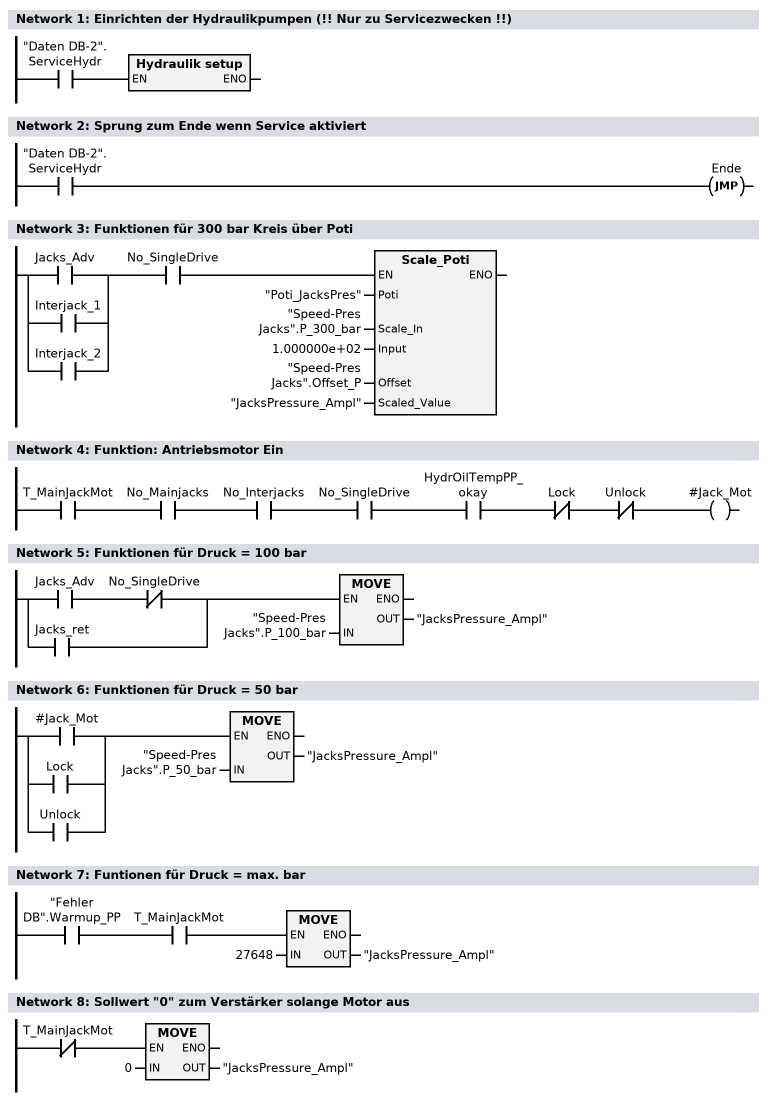
[picture p24: Jacks pressure networks 1-8]
NETWORK
TITLE = Einrichten der Hydraulikpumpen (!! Nur zu Servicezwecken !!)
      A     "Daten DB-2".ServiceHydr;
      JNB   _001;
      CALL  "Hydraulik setup";
_001: NOP   0;
NETWORK
TITLE = Sprung zum Ende wenn Service aktiviert
      A     "Daten DB-2".ServiceHydr;
      JC    Ende;
NETWORK
TITLE = Funktionen für 300 bar Kreis über Poti
      A(;
      O     "Jacks_Adv";
      O     "Interjack_1";
      O     "Interjack_2";
      );
      A     "No_SingleDrive";
      JNB   _002;
      CALL  "Scale_Poti" (
           Poti                     := "Poti_JacksPres",
           Scale_In                 := "Speed-Pres Jacks".P_300_bar,
           Input                    := 1.000000e+02,
           Offset                   := "Speed-Pres Jacks".Offset_P,
           Scaled_Value             := "JacksPressure_Ampl");
_002: NOP   0;
NETWORK
TITLE = Funktion: Antriebsmotor Ein
      A     "T_MainJackMot";
      A     "No_Mainjacks";
      A     "No_Interjacks";
      A     "No_SingleDrive";
      A     "HydrOilTempPP_okay";
      AN    "Lock";
      AN    "Unlock";
      =     #Jack_Mot;
NETWORK
TITLE = Funktionen für Druck = 100 bar
      A(;
      A     "Jacks_Adv";
      AN    "No_SingleDrive";
      O     "Jacks_ret";
      );
      JNB   _003;
      L     "Speed-Pres Jacks".P_100_bar;
      T     "JacksPressure_Ampl";
_003: NOP   0;
NETWORK
TITLE = Funktionen für Druck = 50 bar
      A(;
      O     #Jack_Mot;
      O     "Lock";
      O     "Unlock";
      );
      JNB   _004;
      L     "Speed-Pres Jacks".P_50_bar;
      T     "JacksPressure_Ampl";
_004: NOP   0;
NETWORK
TITLE = Funtionen für Druck = max. bar
      A     "Fehler DB".Warmup_PP;
      A     "T_MainJackMot";
      JNB   _005;
      L     27648;
      T     "JacksPressure_Ampl";
_005: NOP   0;
NETWORK
TITLE = Sollwert "0" zum Verstärker solange Motor aus
      AN    "T_MainJackMot";
      JNB   _006;
      L     0;
      T     "JacksPressure_Ampl";
_006: NOP   0;
NETWORK
TITLE =
Ende: NOP   0;
END_FUNCTION

FUNCTION "Cutter control" : VOID	// FC 25
TITLE = Schürfradsteuerung links/rechts
AUTHOR : Simdon
FAMILY : Cutter
NAME : Cut_Con
VERSION : 0.1
VAR_TEMP
  Mot_okay : BOOL ;	//Antriebsmotor für Hydraulik
  H_Right : BOOL ;
  H_Left : BOOL ;
END_VAR
BEGIN
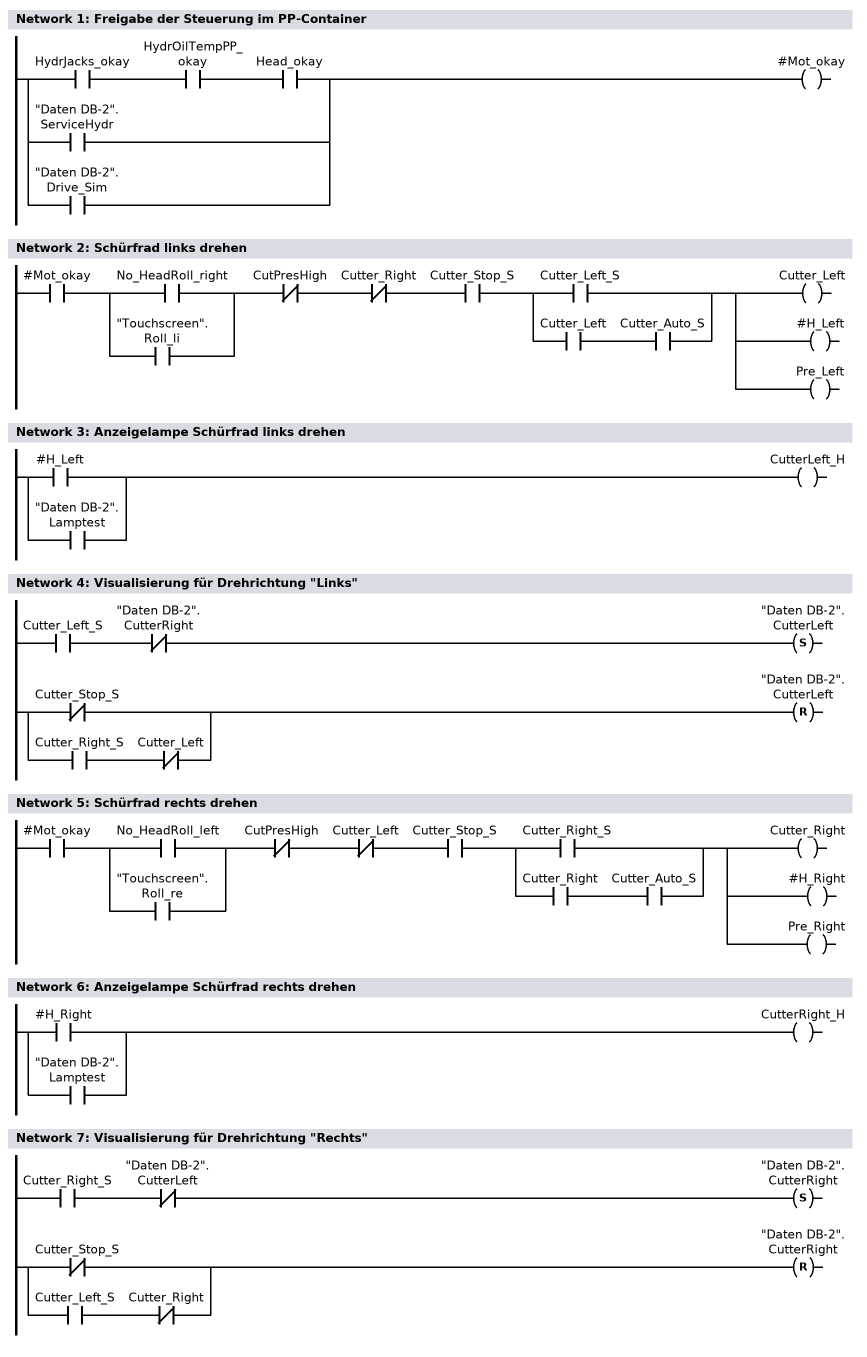
NETWORK
TITLE = Freigabe der Steuerung im PP-Container
      A     "HydrJacks_okay";
      A     "HydrOilTempPP_okay";
      A     "Head_okay";
      O     "Daten DB-2".ServiceHydr;
      O     "Daten DB-2".Drive_Sim;
      =     #Mot_okay;
NETWORK
TITLE = Schürfrad links drehen
//Schürfrad dreht in einer der gewählten Betriebsarten links herum.
      A     #Mot_okay;
      A(;
      O     "No_HeadRoll_right";
      O     "Touchscreen".Roll_li;
      );
      AN    "CutPresHigh";
      AN    "Cutter_Right";
      A     "Cutter_Stop_S";
      A(;
      O     "Cutter_Left_S";
      O;
      A     "Cutter_Left";
      A     "Cutter_Auto_S";
      );
      =     "Cutter_Left";
      =     #H_Left;
      =     "Pre_Left";
NETWORK
TITLE = Anzeigelampe Schürfrad links drehen
      O     #H_Left;
      O     "Daten DB-2".Lamptest;
      =     "CutterLeft_H";
NETWORK
TITLE = Visualisierung für Drehrichtung "Links"
      A     "Cutter_Left_S";
      AN    "Daten DB-2".CutterRight;
      S     "Daten DB-2".CutterLeft;
      A(;
      ON    "Cutter_Stop_S";
      O;
      A     "Cutter_Right_S";
      AN    "Cutter_Left";
      );
      R     "Daten DB-2".CutterLeft;
      NOP   0;
NETWORK
TITLE = Schürfrad rechts drehen
//Schürfrad dreht in einer der gewählten Betriebsarten rechts herum.
      A     #Mot_okay;
      A(;
      O     "No_HeadRoll_left";
      O     "Touchscreen".Roll_re;
      );
      AN    "CutPresHigh";
      AN    "Cutter_Left";
      A     "Cutter_Stop_S";
      A(;
      O     "Cutter_Right_S";
      O;
      A     "Cutter_Right";
      A     "Cutter_Auto_S";
      );
      =     "Cutter_Right";
      =     #H_Right;
      =     "Pre_Right";
NETWORK
TITLE = Anzeigelampe Schürfrad rechts drehen
      O     #H_Right;
      O     "Daten DB-2".Lamptest;
      =     "CutterRight_H";
NETWORK
TITLE = Visualisierung für Drehrichtung "Rechts"
      A     "Cutter_Right_S";
      AN    "Daten DB-2".CutterLeft;
      S     "Daten DB-2".CutterRight;
      A(;
      ON    "Cutter_Stop_S";
      O;
      A     "Cutter_Left_S";
      AN    "Cutter_Right";
      );
      R     "Daten DB-2".CutterRight;
      NOP   0;
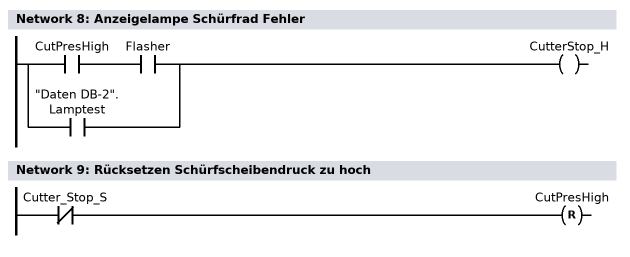
NETWORK
TITLE = Anzeigelampe Schürfrad Fehler
      A     "CutPresHigh";
      A     "Flasher";
      O     "Daten DB-2".Lamptest;
      =     "CutterStop_H";
NETWORK
TITLE = Rücksetzen Schürfscheibendruck zu hoch
      AN    "Cutter_Stop_S";
      R     "CutPresHigh";
END_FUNCTION

FUNCTION "Cutter speed" : VOID	// FC 26
TITLE = Volumenstromeinstellung für Schürfrad im PP-Container
AUTHOR : Simdon
FAMILY : Cutter
NAME : CutVol
VERSION : 0.1
VAR_TEMP
  Ltr_200 : BOOL ;
  Ltr_270 : BOOL ;
  Ltr_max : BOOL ;
END_VAR
BEGIN
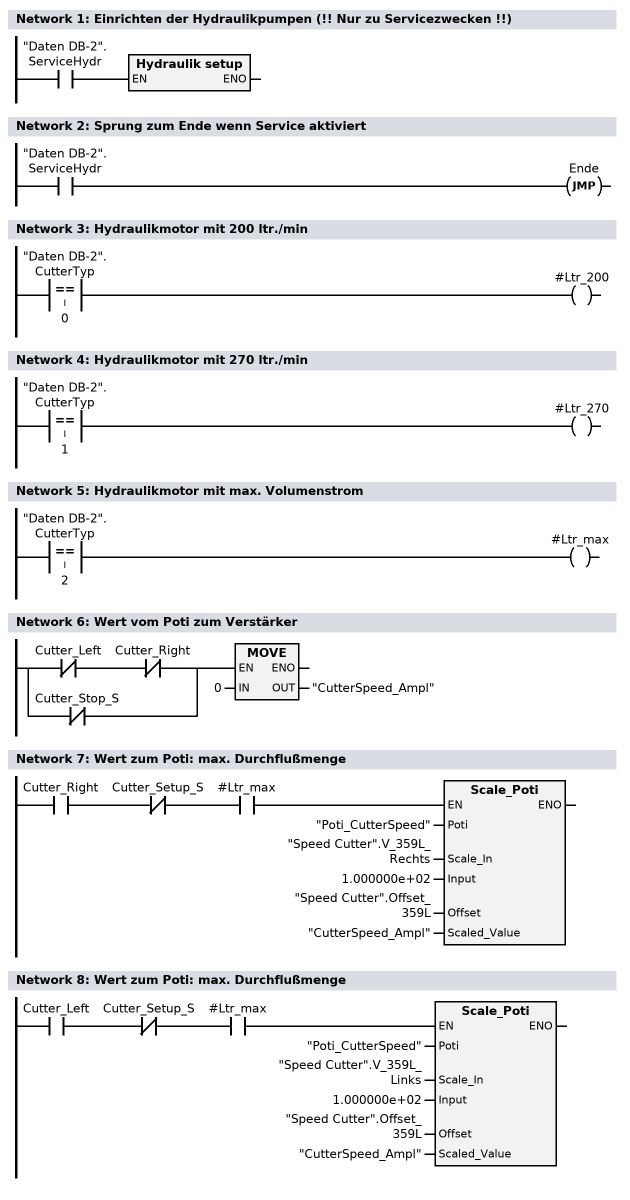
NETWORK
TITLE = Einrichten der Hydraulikpumpen (!! Nur zu Servicezwecken !!)
      A     "Daten DB-2".ServiceHydr;
      JNB   _001;
      CALL  "Hydraulik setup";
_001: NOP   0;
NETWORK
TITLE = Sprung zum Ende wenn Service aktiviert
      A     "Daten DB-2".ServiceHydr;
      JC    Ende;
NETWORK
TITLE = Hydraulikmotor mit 200 ltr./min
      L     "Daten DB-2".CutterTyp;
      L     0;
      ==I;
      =     #Ltr_200;
NETWORK
TITLE = Hydraulikmotor mit 270 ltr./min
      L     "Daten DB-2".CutterTyp;
      L     1;
      ==I;
      =     #Ltr_270;
NETWORK
TITLE = Hydraulikmotor mit max. Volumenstrom
      L     "Daten DB-2".CutterTyp;
      L     2;
      ==I;
      =     #Ltr_max;
NETWORK
TITLE = Wert vom Poti zum Verstärker
      A(;
      AN    "Cutter_Left";
      AN    "Cutter_Right";
      ON    "Cutter_Stop_S";
      );
      JNB   _002;
      L     0;
      T     "CutterSpeed_Ampl";
_002: NOP   0;
NETWORK
TITLE = Wert zum Poti: max. Durchflußmenge
      A     "Cutter_Right";
      AN    "Cutter_Setup_S";
      A     #Ltr_max;
      JNB   _003;
      CALL  "Scale_Poti" (
           Poti                     := "Poti_CutterSpeed",
           Scale_In                 := "Speed Cutter".V_359L_Rechts,
           Input                    := 1.000000e+02,
           Offset                   := "Speed Cutter".Offset_359L,
           Scaled_Value             := "CutterSpeed_Ampl");
_003: NOP   0;
NETWORK
TITLE = Wert zum Poti: max. Durchflußmenge
      A     "Cutter_Left";
      AN    "Cutter_Setup_S";
      A     #Ltr_max;
      JNB   _004;
      CALL  "Scale_Poti" (
           Poti                     := "Poti_CutterSpeed",
           Scale_In                 := "Speed Cutter".V_359L_Links,
           Input                    := 1.000000e+02,
           Offset                   := "Speed Cutter".Offset_359L,
           Scaled_Value             := "CutterSpeed_Ampl");
_004: NOP   0;
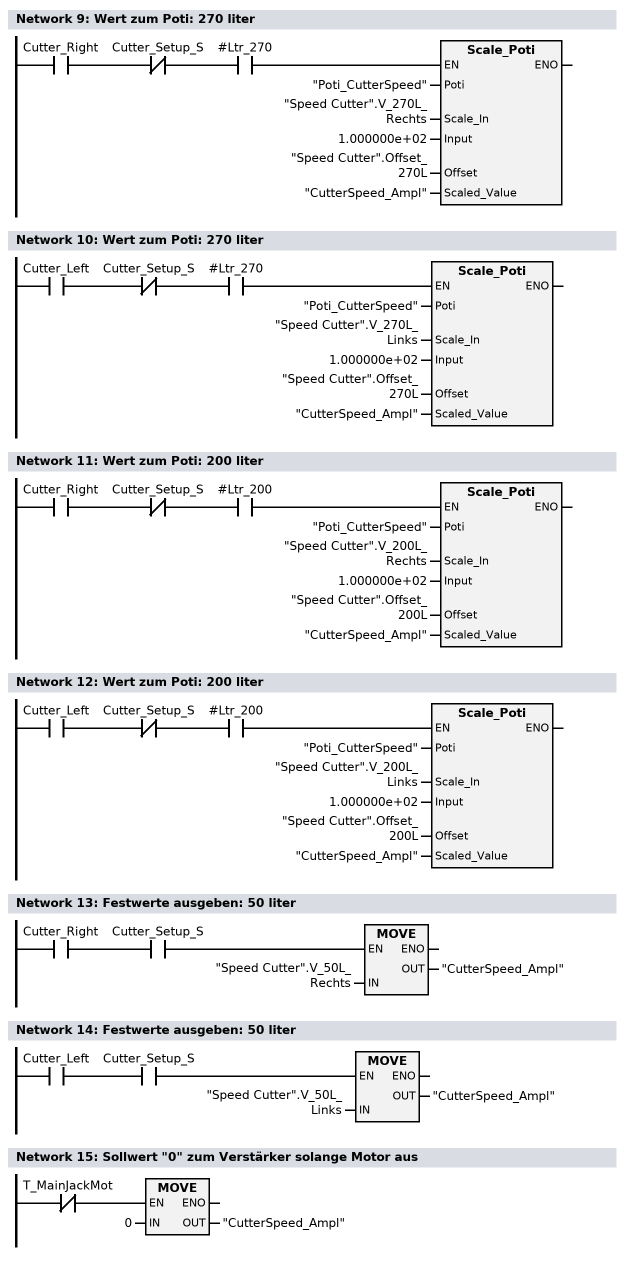
NETWORK
TITLE = Wert zum Poti: 270 liter
      A     "Cutter_Right";
      AN    "Cutter_Setup_S";
      A     #Ltr_270;
      JNB   _005;
      CALL  "Scale_Poti" (
           Poti                     := "Poti_CutterSpeed",
           Scale_In                 := "Speed Cutter".V_270L_Rechts,
           Input                    := 1.000000e+02,
           Offset                   := "Speed Cutter".Offset_270L,
           Scaled_Value             := "CutterSpeed_Ampl");
_005: NOP   0;
NETWORK
TITLE = Wert zum Poti: 270 liter
      A     "Cutter_Left";
      AN    "Cutter_Setup_S";
      A     #Ltr_270;
      JNB   _006;
      CALL  "Scale_Poti" (
           Poti                     := "Poti_CutterSpeed",
           Scale_In                 := "Speed Cutter".V_270L_Links,
           Input                    := 1.000000e+02,
           Offset                   := "Speed Cutter".Offset_270L,
           Scaled_Value             := "CutterSpeed_Ampl");
_006: NOP   0;
NETWORK
TITLE = Wert zum Poti: 200 liter
      A     "Cutter_Right";
      AN    "Cutter_Setup_S";
      A     #Ltr_200;
      JNB   _007;
      CALL  "Scale_Poti" (
           Poti                     := "Poti_CutterSpeed",
           Scale_In                 := "Speed Cutter".V_200L_Rechts,
           Input                    := 1.000000e+02,
           Offset                   := "Speed Cutter".Offset_200L,
           Scaled_Value             := "CutterSpeed_Ampl");
_007: NOP   0;
NETWORK
TITLE = Wert zum Poti: 200 liter
      A     "Cutter_Left";
      AN    "Cutter_Setup_S";
      A     #Ltr_200;
      JNB   _008;
      CALL  "Scale_Poti" (
           Poti                     := "Poti_CutterSpeed",
           Scale_In                 := "Speed Cutter".V_200L_Links,
           Input                    := 1.000000e+02,
           Offset                   := "Speed Cutter".Offset_200L,
           Scaled_Value             := "CutterSpeed_Ampl");
_008: NOP   0;
NETWORK
TITLE = Festwerte ausgeben: 50 liter
      A     "Cutter_Right";
      A     "Cutter_Setup_S";
      JNB   _009;
      L     "Speed Cutter".V_50L_Rechts;
      T     "CutterSpeed_Ampl";
_009: NOP   0;
NETWORK
TITLE = Festwerte ausgeben: 50 liter
      A     "Cutter_Left";
      A     "Cutter_Setup_S";
      JNB   _00a;
      L     "Speed Cutter".V_50L_Links;
      T     "CutterSpeed_Ampl";
_00a: NOP   0;
NETWORK
TITLE = Sollwert "0" zum Verstärker solange Motor aus
      AN    "T_MainJackMot";
      JNB   _00b;
      L     0;
      T     "CutterSpeed_Ampl";
_00b: NOP   0;
NETWORK
TITLE = Bausteinende
Ende: NOP   0;
END_FUNCTION

FUNCTION "Valve control" : VOID	// FC 29
TITLE = Allgemeine Ventilansteuerung für die mts1000
AUTHOR : Simdon
FAMILY : Hydrauli
NAME : ValveCon
VERSION : 0.1
BEGIN
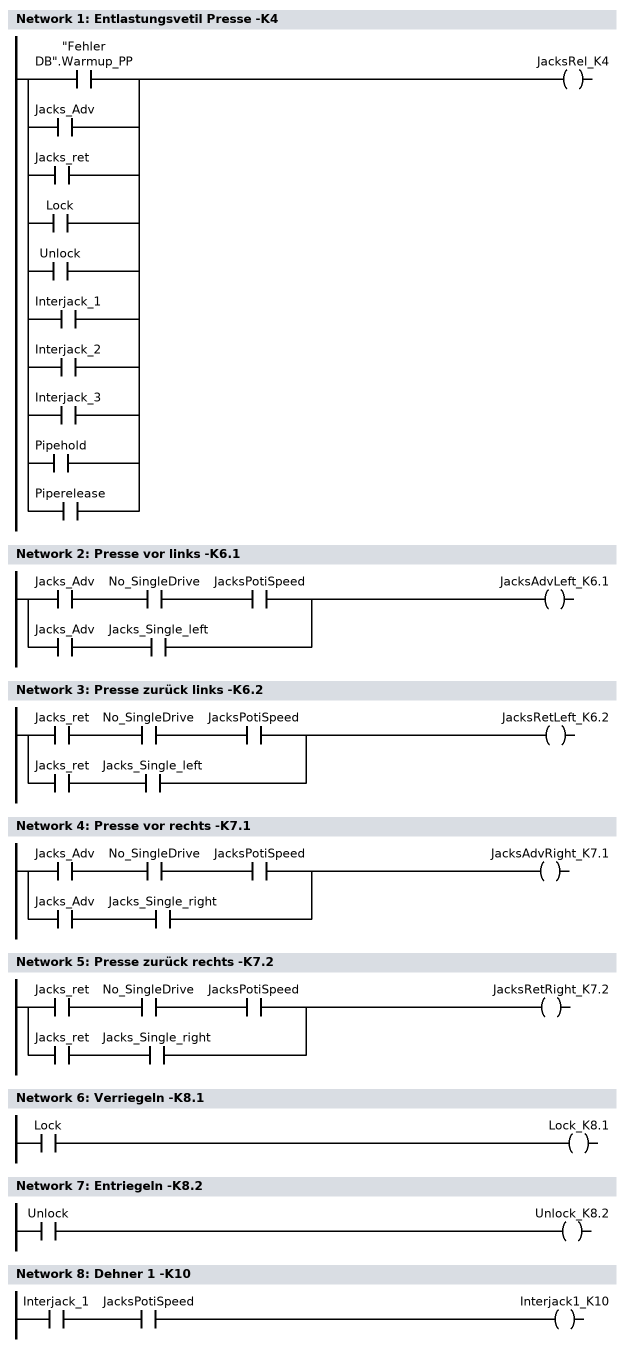
NETWORK
TITLE = Entlastungsvetil Presse -K4
      O     "Fehler DB".Warmup_PP;
      O     "Jacks_Adv";
      O     "Jacks_ret";
      O     "Lock";
      O     "Unlock";
      O     "Interjack_1";
      O     "Interjack_2";
      O     "Interjack_3";
      O     "Pipehold";
      O     "Piperelease";
      =     "JacksRel_K4";
NETWORK
TITLE = Presse vor links -K6.1
      A     "Jacks_Adv";
      A     "No_SingleDrive";
      A     "JacksPotiSpeed";
      O;
      A     "Jacks_Adv";
      A     "Jacks_Single_left";
      =     "JacksAdvLeft_K6.1";
NETWORK
TITLE = Presse zurück links -K6.2
      A     "Jacks_ret";
      A     "No_SingleDrive";
      A     "JacksPotiSpeed";
      O;
      A     "Jacks_ret";
      A     "Jacks_Single_left";
      =     "JacksRetLeft_K6.2";
NETWORK
TITLE = Presse vor rechts -K7.1
      A     "Jacks_Adv";
      A     "No_SingleDrive";
      A     "JacksPotiSpeed";
      O;
      A     "Jacks_Adv";
      A     "Jacks_Single_right";
      =     "JacksAdvRight_K7.1";
NETWORK
TITLE = Presse zurück rechts -K7.2
      A     "Jacks_ret";
      A     "No_SingleDrive";
      A     "JacksPotiSpeed";
      O;
      A     "Jacks_ret";
      A     "Jacks_Single_right";
      =     "JacksRetRight_K7.2";
NETWORK
TITLE = Verriegeln -K8.1
      A     "Lock";
      =     "Lock_K8.1";
NETWORK
TITLE = Entriegeln -K8.2
      A     "Unlock";
      =     "Unlock_K8.2";
NETWORK
TITLE = Dehner 1 -K10
      A     "Interjack_1";
      A     "JacksPotiSpeed";
      =     "Interjack1_K10";
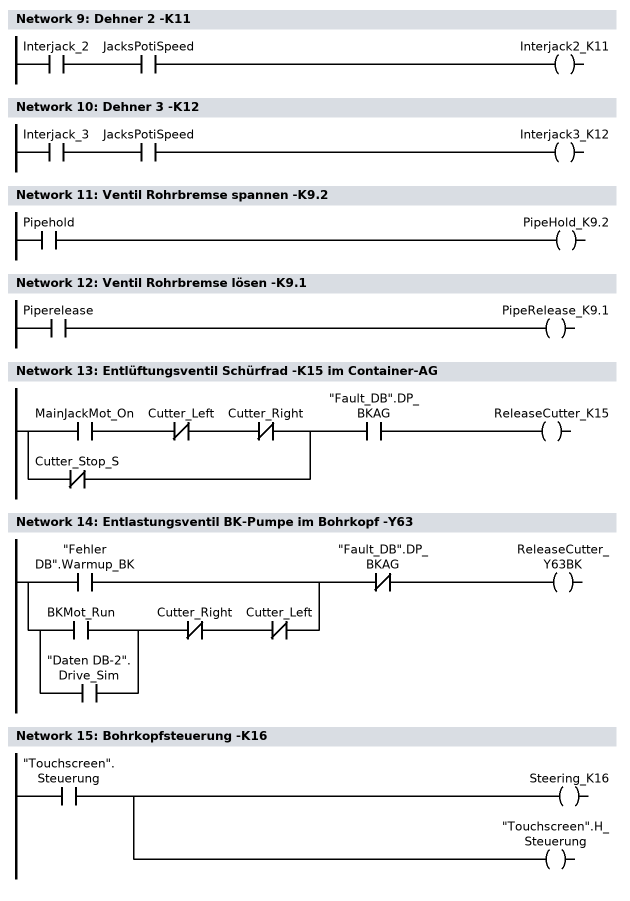
NETWORK
TITLE = Dehner 2 -K11
      A     "Interjack_2";
      A     "JacksPotiSpeed";
      =     "Interjack2_K11";
NETWORK
TITLE = Dehner 3 -K12
      A     "Interjack_3";
      A     "JacksPotiSpeed";
      =     "Interjack3_K12";
NETWORK
TITLE = Ventil Rohrbremse spannen -K9.2
      A     "Pipehold";
      =     "PipeHold_K9.2";
NETWORK
TITLE = Ventil Rohrbremse lösen -K9.1
      A     "Piperelease";
      =     "PipeRelease_K9.1";
NETWORK
TITLE = Entlüftungsventil Schürfrad -K15 im Container-AG
      A(;
      A     "MainJackMot_On";
      AN    "Cutter_Left";
      AN    "Cutter_Right";
      ON    "Cutter_Stop_S";
      );
      A     "Fault_DB".DP_BKAG;
      =     "ReleaseCutter_K15";
NETWORK
TITLE = Entlastungsventil BK-Pumpe im Bohrkopf -Y63
      A(;
      O     "Fehler DB".Warmup_BK;
      O;
      A(;
      O     "BKMot_Run";
      O     "Daten DB-2".Drive_Sim;
      );
      AN    "Cutter_Right";
      AN    "Cutter_Left";
      );
      AN    "Fault_DB".DP_BKAG;
      =     "ReleaseCutter_Y63BK";
NETWORK
TITLE = Bohrkopfsteuerung -K16
      A     "Touchscreen".Steuerung;
      =     "Steering_K16";
      =     "Touchscreen".H_Steuerung;
END_FUNCTION

FUNCTION "Hydraulic power pack" : VOID	// FC 30
TITLE = Hydraulikölstand-und Temperatur Aggregat (Container) Fan1
AUTHOR : Simdon
FAMILY : Freigabe
NAME : Hydr_PP
VERSION : 0.1
VAR_TEMP
  PresSens : BOOL ;	//Fehler Drucksensor
  Feedlinefilter : REAL ;
  DelayFilter : BOOL ;
  RetVal_1 : BOOL ;
  RetVal_2 : BOOL ;
END_VAR
BEGIN
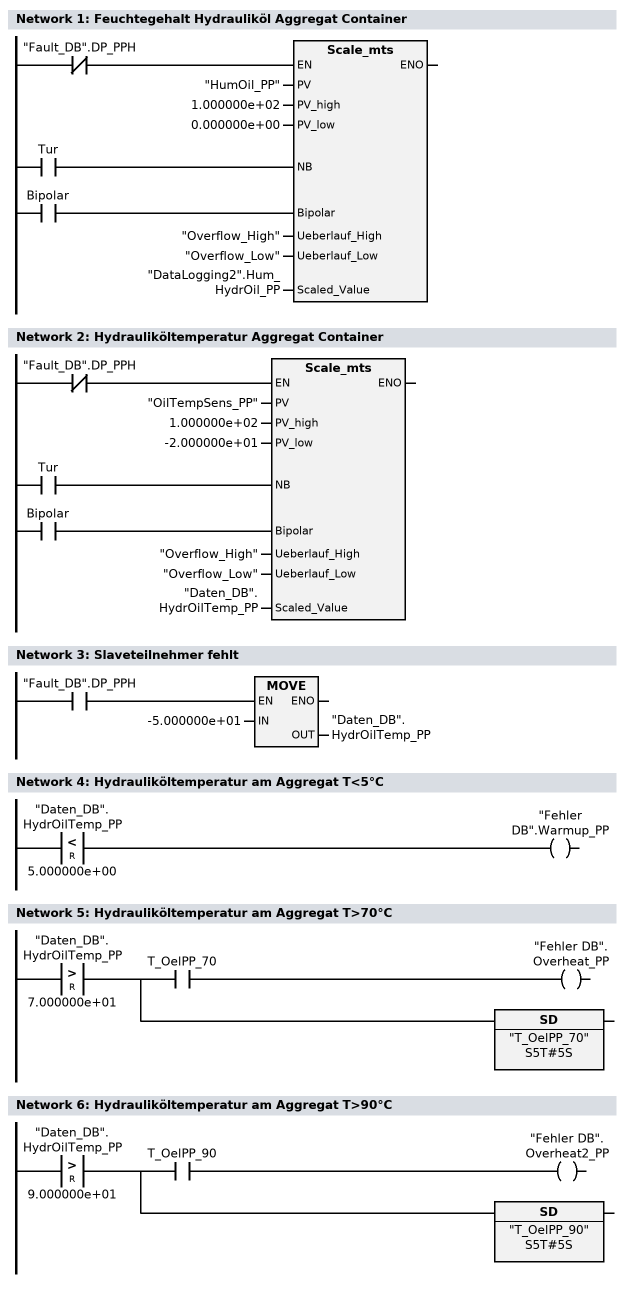
NETWORK
TITLE = Feuchtegehalt Hydrauliköl Aggregat Container
//Im FC21 werden die Werte des Temperatur-Sensors eingelesen und als skalierte 
//Werte in den Grenzen zwischen -50°C und 200°C ausgegeben.
      A     "Tur";
      =     L 7.0;
      BLD   103;
      A     "Bipolar";
      =     L 7.1;
      BLD   103;
      AN    "Fault_DB".DP_PPH;
      JNB   _001;
      CALL  "Scale_mts" (
           PV                       := "HumOil_PP",
           PV_high                  := 1.000000e+02,
           PV_low                   := 0.000000e+00,
           NB                       := L 7.0,
           Bipolar                  := L 7.1,
           Ueberlauf_High           := "Overflow_High",
           Ueberlauf_Low            := "Overflow_Low",
           Scaled_Value             := "DataLogging2".Hum_HydrOil_PP);
_001: NOP   0;
NETWORK
TITLE = Hydrauliköltemperatur Aggregat Container
//Im FC21 werden die Werte des Temperatur-Sensors eingelesen und als skalierte 
//Werte in den Grenzen zwischen -50°C und 200°C ausgegeben.
      A     "Tur";
      =     L 7.0;
      BLD   103;
      A     "Bipolar";
      =     L 7.1;
      BLD   103;
      AN    "Fault_DB".DP_PPH;
      JNB   _002;
      CALL  "Scale_mts" (
           PV                       := "OilTempSens_PP",
           PV_high                  := 1.000000e+02,
           PV_low                   := -2.000000e+01,
           NB                       := L 7.0,
           Bipolar                  := L 7.1,
           Ueberlauf_High           := "Overflow_High",
           Ueberlauf_Low            := "Overflow_Low",
           Scaled_Value             := "Daten_DB".HydrOilTemp_PP);
_002: NOP   0;
NETWORK
TITLE = Slaveteilnehmer fehlt
      A     "Fault_DB".DP_PPH;
      JNB   _003;
      L     -5.000000e+01;
      T     "Daten_DB".HydrOilTemp_PP;
_003: NOP   0;
NETWORK
TITLE = Hydrauliköltemperatur am Aggregat T<5°C
//Datendoppelwort DB10.dbd16 (Hydrauliköltemperatur) wird verglichen mit dem Wert 
//"5", um herauszufinden, ob es kleiner ist. 
//Ist es kleiner wird der Merker 15.3 auf "TRUE" gesetzt.
      L     "Daten_DB".HydrOilTemp_PP;
      L     5.000000e+00;
      <R;
      =     "Fehler DB".Warmup_PP;
NETWORK
TITLE = Hydrauliköltemperatur am Aggregat T>70°C
//Datendoppelwort DB10.dbd16 (Hydrauliköltemperatur) wird verglichen mit dem Wert 
//"70", um herauszufinden, ob es größer ist.
//Ist es größer wird der Merker 15.4 auf "TRUE" gesetzt.
      L     "Daten_DB".HydrOilTemp_PP;
      L     7.000000e+01;
      >R;
      =     L 7.0;
      A     L 7.0;
      A     "T_OelPP_70";
      =     "Fehler DB".Overheat_PP;
      A     L 7.0;
      BLD   102;
      L     S5T#5S;
      SD    "T_OelPP_70";
NETWORK
TITLE = Hydrauliköltemperatur am Aggregat T>90°C
//Datendoppelwort DB10.dbd16 (Hydrauliköltemperatur) wird verglichen mit dem Wert 
//"70", um herauszufinden, ob es größer ist.
//Ist es größer wird der Merker 15.4 auf "TRUE" gesetzt.
      L     "Daten_DB".HydrOilTemp_PP;
      L     9.000000e+01;
      >R;
      =     L 7.0;
      A     L 7.0;
      A     "T_OelPP_90";
      =     "Fehler DB".Overheat2_PP;
      A     L 7.0;
      BLD   102;
      L     S5T#5S;
      SD    "T_OelPP_90";
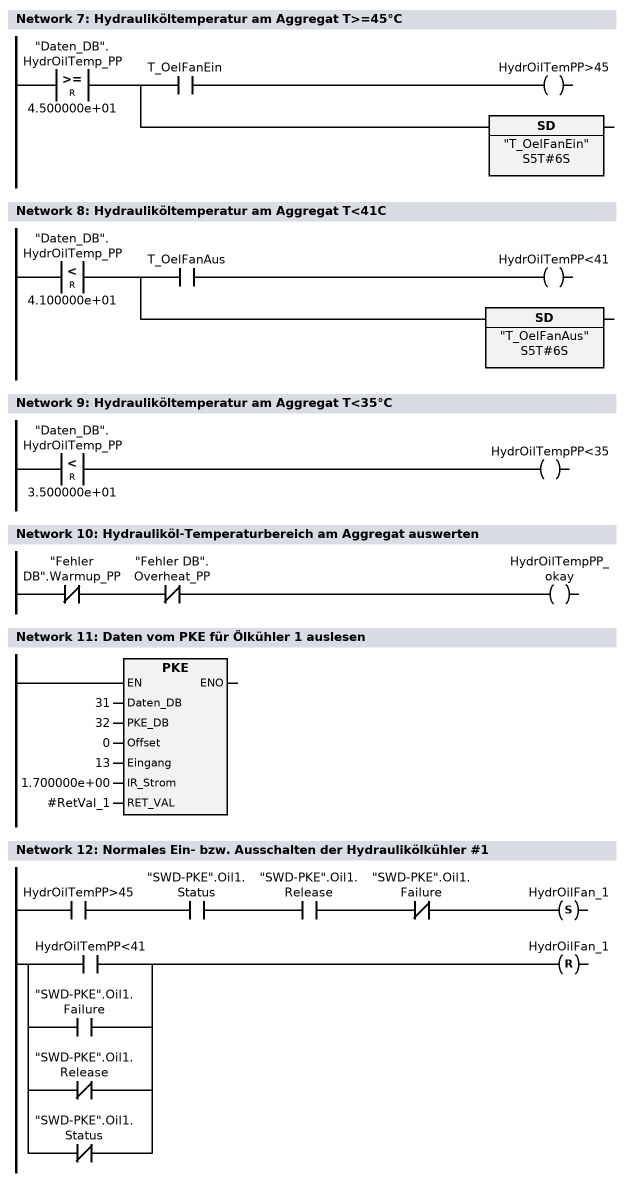
NETWORK
TITLE = Hydrauliköltemperatur am Aggregat T>=45°C
//Datendoppelwort DB10.dbd16 (Hydrauliköltemperatur) wird verglichen mit dem Wert 
//"38", um herauszufinden, ob es größer ist.
//Ist es größer wird der Merker 15.5 auf "TRUE" gesetzt.
      L     "Daten_DB".HydrOilTemp_PP;
      L     4.500000e+01;
      >=R;
      =     L 7.0;
      A     L 7.0;
      A     "T_OelFanEin";
      =     "HydrOilTemPP>45";
      A     L 7.0;
      BLD   102;
      L     S5T#6S;
      SD    "T_OelFanEin";
NETWORK
TITLE = Hydrauliköltemperatur am Aggregat T<41C
//Datendoppelwort DB10.dbd16 (Hydrauliköltemperatur) wird verglichen mit dem Wert 
//"35", um herauszufinden, ob es größer ist.
//Ist es kleiner wird der Merker 16 auf "TRUE" gesetzt.
      L     "Daten_DB".HydrOilTemp_PP;
      L     4.100000e+01;
      <R;
      =     L 7.0;
      A     L 7.0;
      A     "T_OelFanAus";
      =     "HydrOilTemPP<41";
      A     L 7.0;
      BLD   102;
      L     S5T#6S;
      SD    "T_OelFanAus";
NETWORK
TITLE = Hydrauliköltemperatur am Aggregat T<35°C
//Datendoppelwort DB10.dbd16 (Hydrauliköltemperatur) wird verglichen mit dem Wert 
//"35", um herauszufinden, ob es größer ist.
//Ist es kleiner wird der Merker 16 auf "TRUE" gesetzt.
      L     "Daten_DB".HydrOilTemp_PP;
      L     3.500000e+01;
      <R;
      =     "HydrOilTempPP<35";
NETWORK
TITLE = Hydrauliköl-Temperaturbereich am Aggregat auswerten
//Liegt der Hydrauliköl-Temperaturbereich am Aggregat zwischen 5°C und 70°C wird
//der Merker 15.2 gesetzt.
      AN    "Fehler DB".Warmup_PP;
      AN    "Fehler DB".Overheat_PP;
      =     "HydrOilTempPP_okay";
NETWORK
TITLE = Daten vom PKE für Ölkühler 1 auslesen
      CALL  "PKE" (
           Daten_DB                 := 31,
           PKE_DB                   := 32,
           Offset                   := 0,
           Eingang                  := 13,
           IR_Strom                 := 1.700000e+00,
           RET_VAL                  := #RetVal_1);
      NOP   0;
NETWORK
TITLE = Normales Ein- bzw. Ausschalten der Hydraulikölkühler #1
      A     "HydrOilTemPP>45";
      A     "SWD-PKE".Oil1.Status;
      A     "SWD-PKE".Oil1.Release;
      AN    "SWD-PKE".Oil1.Failure;
      S     "HydrOilFan_1";
      A(;
      O     "HydrOilTemPP<41";
      O     "SWD-PKE".Oil1.Failure;
      ON    "SWD-PKE".Oil1.Release;
      ON    "SWD-PKE".Oil1.Status;
      );
      R     "HydrOilFan_1";
      NOP   0;
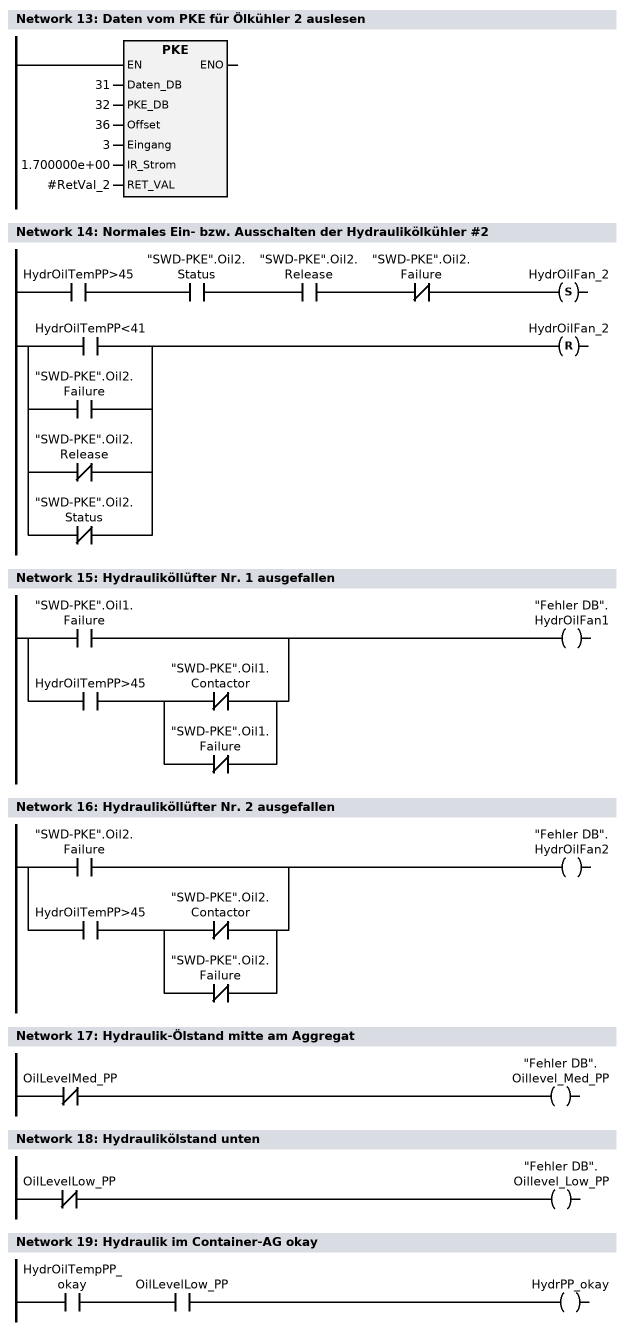
NETWORK
TITLE = Daten vom PKE für Ölkühler 2 auslesen
      CALL  "PKE" (
           Daten_DB                 := 31,
           PKE_DB                   := 32,
           Offset                   := 36,
           Eingang                  := 3,
           IR_Strom                 := 1.700000e+00,
           RET_VAL                  := #RetVal_2);
      NOP   0;
NETWORK
TITLE = Normales Ein- bzw. Ausschalten der Hydraulikölkühler #2
      A     "HydrOilTemPP>45";
      A     "SWD-PKE".Oil2.Status;
      A     "SWD-PKE".Oil2.Release;
      AN    "SWD-PKE".Oil2.Failure;
      S     "HydrOilFan_2";
      A(;
      O     "HydrOilTemPP<41";
      O     "SWD-PKE".Oil2.Failure;
      ON    "SWD-PKE".Oil2.Release;
      ON    "SWD-PKE".Oil2.Status;
      );
      R     "HydrOilFan_2";
      NOP   0;
NETWORK
TITLE = Hydrauliköllüfter Nr. 1 ausgefallen
      O     "SWD-PKE".Oil1.Failure;
      O;
      A     "HydrOilTemPP>45";
      A(;
      ON    "SWD-PKE".Oil1.Contactor;
      ON    "SWD-PKE".Oil1.Failure;
      );
      =     "Fehler DB".HydrOilFan1;
NETWORK
TITLE = Hydrauliköllüfter Nr. 2 ausgefallen
      O     "SWD-PKE".Oil2.Failure;
      O;
      A     "HydrOilTemPP>45";
      A(;
      ON    "SWD-PKE".Oil2.Contactor;
      ON    "SWD-PKE".Oil2.Failure;
      );
      =     "Fehler DB".HydrOilFan2;
NETWORK
TITLE = Hydraulik-Ölstand mitte am Aggregat
//Bei Hydraulik-Ölstand mitte am Aggregat öffnet der Oellevel-Schalter mitte 
//und der Merker M14.7 wird gesetzt. 
      AN    "OilLevelMed_PP";
      =     "Fehler DB".Oillevel_Med_PP;
NETWORK
TITLE = Hydraulikölstand unten
//Bei Hydraulik-Ölstand unten am Aggregat öffnet der Oellevel-Schalter unten 
//und der Merker M15.0 wird gesetzt.
      AN    "OilLevelLow_PP";
      =     "Fehler DB".Oillevel_Low_PP;
NETWORK
TITLE = Hydraulik im Container-AG okay
      A     "HydrOilTempPP_okay";
      A     "OilLevelLow_PP";
      =     "HydrPP_okay";
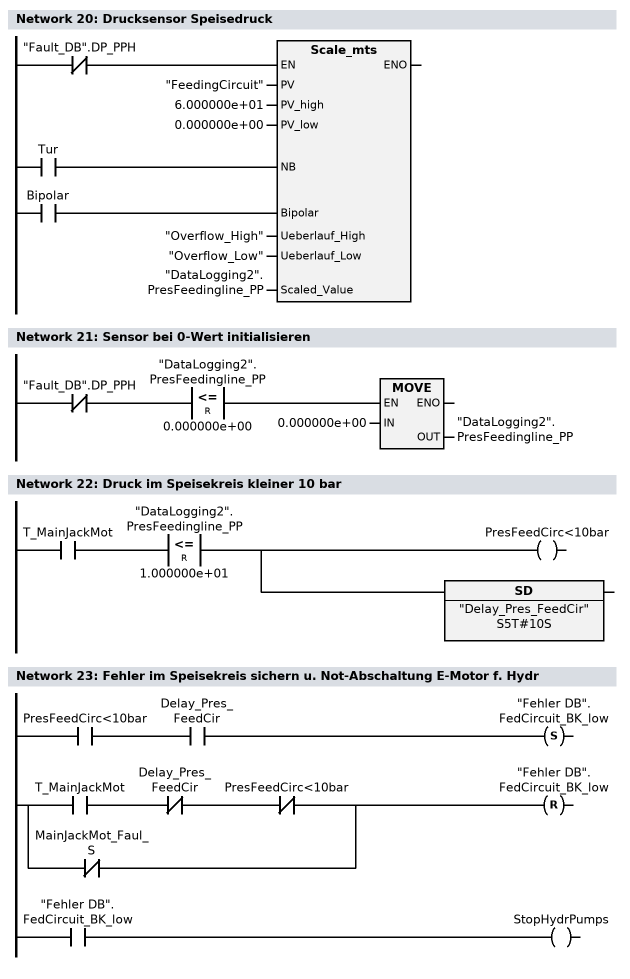
NETWORK
TITLE = Drucksensor Speisedruck
      A     "Tur";
      =     L 7.0;
      BLD   103;
      A     "Bipolar";
      =     L 7.1;
      BLD   103;
      AN    "Fault_DB".DP_PPH;
      JNB   _004;
      CALL  "Scale_mts" (
           PV                       := "FeedingCircuit",
           PV_high                  := 6.000000e+01,
           PV_low                   := 0.000000e+00,
           NB                       := L 7.0,
           Bipolar                  := L 7.1,
           Ueberlauf_High           := "Overflow_High",
           Ueberlauf_Low            := "Overflow_Low",
           Scaled_Value             := "DataLogging2".PresFeedingline_PP);
_004: NOP   0;
NETWORK
TITLE = Sensor bei 0-Wert initialisieren
      AN    "Fault_DB".DP_PPH;
      A(;
      L     "DataLogging2".PresFeedingline_PP;
      L     0.000000e+00;
      <=R;
      );
      JNB   _005;
      L     0.000000e+00;
      T     "DataLogging2".PresFeedingline_PP;
_005: NOP   0;
NETWORK
TITLE = Druck im Speisekreis kleiner 10 bar
      A     "T_MainJackMot";
      A(;
      L     "DataLogging2".PresFeedingline_PP;
      L     1.000000e+01;
      <=R;
      );
      =     "PresFeedCirc<10bar";
      L     S5T#10S;
      SD    "Delay_Pres_FeedCir";
NETWORK
TITLE = Fehler im Speisekreis sichern u. Not-Abschaltung E-Motor f. Hydr
      A     "PresFeedCirc<10bar";
      A     "Delay_Pres_FeedCir";
      S     "Fehler DB".FedCircuit_BK_low;
      A(;
      A     "T_MainJackMot";
      AN    "Delay_Pres_FeedCir";
      AN    "PresFeedCirc<10bar";
      ON    "MainJackMot_Faul_S";
      );
      R     "Fehler DB".FedCircuit_BK_low;
      A     "Fehler DB".FedCircuit_BK_low;
      =     "StopHydrPumps";
END_FUNCTION

FUNCTION "Hydraulic_BK" : VOID	// FC 31
TITLE = Hydraulikölstand-und Temperatur im Bohrkopfaggregat
AUTHOR : Simdon
FAMILY : Freigabe
NAME : Hydr_BK
VERSION : 0.1
VAR_TEMP
  Ret1 : WORD ;
END_VAR
BEGIN
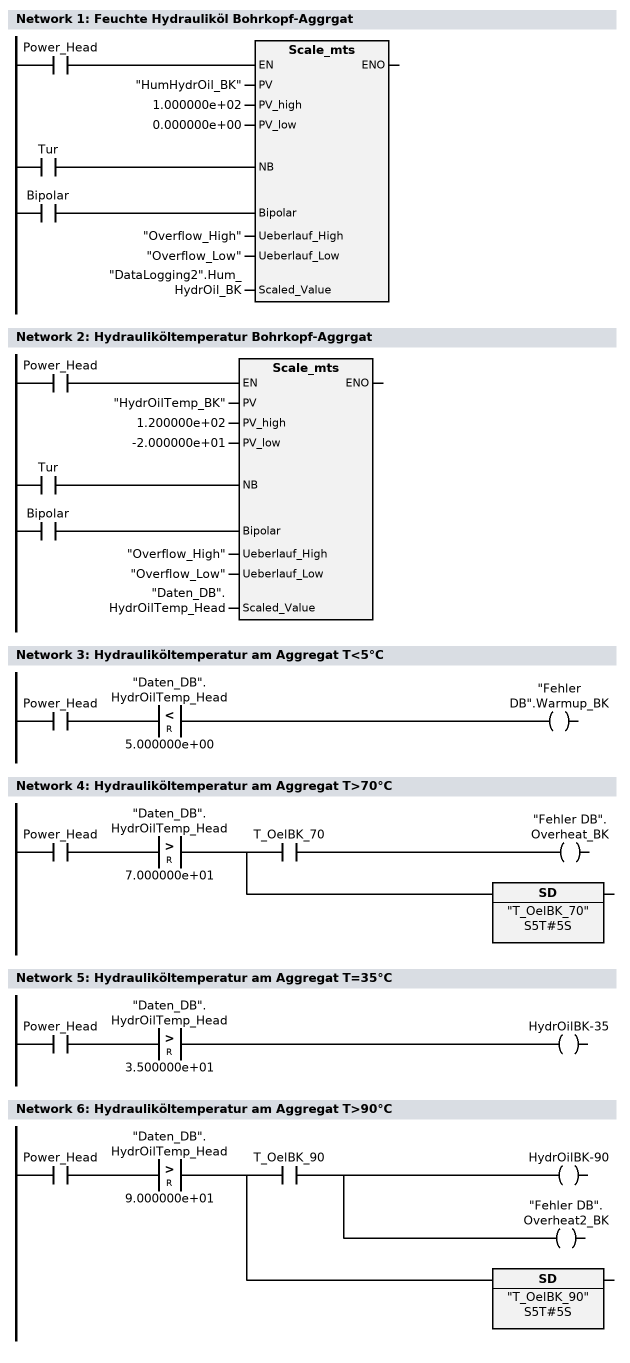
NETWORK
TITLE = Feuchte Hydrauliköl Bohrkopf-Aggrgat
//Im FC21 werden die Werte des Temperatur-Sensors eingelesen und als skalierte 
//Werte in den Grenzen zwischen -50°C und 200°C ausgegeben.
      A     "Tur";
      =     L 2.0;
      BLD   103;
      A     "Bipolar";
      =     L 2.1;
      BLD   103;
      A     "Power_Head";
      JNB   _001;
      CALL  "Scale_mts" (
           PV                       := "HumHydrOil_BK",
           PV_high                  := 1.000000e+02,
           PV_low                   := 0.000000e+00,
           NB                       := L 2.0,
           Bipolar                  := L 2.1,
           Ueberlauf_High           := "Overflow_High",
           Ueberlauf_Low            := "Overflow_Low",
           Scaled_Value             := "DataLogging2".Hum_HydrOil_BK);
_001: NOP   0;
NETWORK
TITLE = Hydrauliköltemperatur Bohrkopf-Aggrgat
//Im FC21 werden die Werte des Temperatur-Sensors eingelesen und als skalierte 
//Werte in den Grenzen zwischen -50°C und 200°C ausgegeben.
      A     "Tur";
      =     L 2.0;
      BLD   103;
      A     "Bipolar";
      =     L 2.1;
      BLD   103;
      A     "Power_Head";
      JNB   _002;
      CALL  "Scale_mts" (
           PV                       := "HydrOilTemp_BK",
           PV_high                  := 1.200000e+02,
           PV_low                   := -2.000000e+01,
           NB                       := L 2.0,
           Bipolar                  := L 2.1,
           Ueberlauf_High           := "Overflow_High",
           Ueberlauf_Low            := "Overflow_Low",
           Scaled_Value             := "Daten_DB".HydrOilTemp_Head);
_002: NOP   0;
NETWORK
TITLE = Hydrauliköltemperatur am Aggregat T<5°C
//Datendoppelwort DB10.dbd16 (Hydrauliköltemperatur) wird verglichen mit dem Wert 
//"5", um herauszufinden, ob es kleiner ist. 
//Ist es kleiner wird der Merker 15.3 auf "TRUE" gesetzt.
      A     "Power_Head";
      A(;
      L     "Daten_DB".HydrOilTemp_Head;
      L     5.000000e+00;
      <R;
      );
      =     "Fehler DB".Warmup_BK;
NETWORK
TITLE = Hydrauliköltemperatur am Aggregat T>70°C
//Datendoppelwort DB10.dbd16 (Hydrauliköltemperatur) wird verglichen mit dem Wert 
//"70", um herauszufinden, ob es größer ist.
//Ist es größer wird der Merker 15.4 auf "TRUE" gesetzt.
      A     "Power_Head";
      A(;
      L     "Daten_DB".HydrOilTemp_Head;
      L     7.000000e+01;
      >R;
      );
      =     L 2.0;
      A     L 2.0;
      A     "T_OelBK_70";
      =     "Fehler DB".Overheat_BK;
      A     L 2.0;
      BLD   102;
      L     S5T#5S;
      SD    "T_OelBK_70";
NETWORK
TITLE = Hydrauliköltemperatur am Aggregat T=35°C
//Datendoppelwort DB10.dbd16 (Hydrauliköltemperatur) wird verglichen mit dem Wert 
//"70", um herauszufinden, ob es größer ist.
//Ist es größer wird der Merker 15.4 auf "TRUE" gesetzt.
      A     "Power_Head";
      A(;
      L     "Daten_DB".HydrOilTemp_Head;
      L     3.500000e+01;
      >R;
      );
      =     "HydrOilBK-35";
NETWORK
TITLE = Hydrauliköltemperatur am Aggregat T>90°C
//Datendoppelwort DB10.dbd16 (Hydrauliköltemperatur) wird verglichen mit dem Wert 
//"70", um herauszufinden, ob es größer ist.
//Ist es größer wird der Merker 15.4 auf "TRUE" gesetzt.
      A     "Power_Head";
      A(;
      L     "Daten_DB".HydrOilTemp_Head;
      L     9.000000e+01;
      >R;
      );
      =     L 2.0;
      A     L 2.0;
      A     "T_OelBK_90";
      =     "HydrOilBK-90";
      =     "Fehler DB".Overheat2_BK;
      A     L 2.0;
      BLD   102;
      L     S5T#5S;
      SD    "T_OelBK_90";
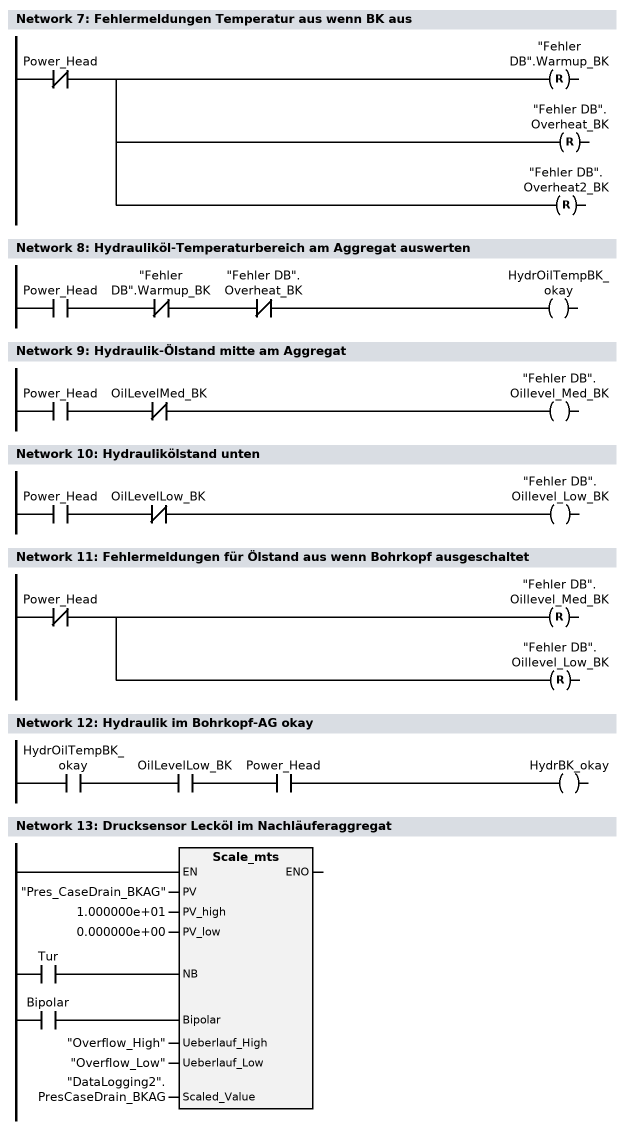
NETWORK
TITLE = Fehlermeldungen Temperatur aus wenn BK aus
      AN    "Power_Head";
      R     "Fehler DB".Warmup_BK;
      R     "Fehler DB".Overheat_BK;
      R     "Fehler DB".Overheat2_BK;
NETWORK
TITLE = Hydrauliköl-Temperaturbereich am Aggregat auswerten
//Liegt der Hydrauliköl-Temperaturbereich am Aggregat zwischen 5°C und 70°C wird
//der Merker 15.2 gesetzt.
      A     "Power_Head";
      AN    "Fehler DB".Warmup_BK;
      AN    "Fehler DB".Overheat_BK;
      =     "HydrOilTempBK_okay";
NETWORK
TITLE = Hydraulik-Ölstand mitte am Aggregat
//Bei Hydraulik-Ölstand mitte am Aggregat öffnet der Oellevel-Schalter mitte 
//und der Merker M14.7 wird gesetzt. 
      A     "Power_Head";
      AN    "OilLevelMed_BK";
      =     "Fehler DB".Oillevel_Med_BK;
NETWORK
TITLE = Hydraulikölstand unten
//Bei Hydraulik-Ölstand unten am Aggregat öffnet der Oellevel-Schalter unten 
//und der Merker M15.0 wird gesetzt.
      A     "Power_Head";
      AN    "OilLevelLow_BK";
      =     "Fehler DB".Oillevel_Low_BK;
NETWORK
TITLE = Fehlermeldungen für Ölstand aus wenn Bohrkopf ausgeschaltet
      AN    "Power_Head";
      R     "Fehler DB".Oillevel_Med_BK;
      R     "Fehler DB".Oillevel_Low_BK;
NETWORK
TITLE = Hydraulik im Bohrkopf-AG okay
      A     "HydrOilTempBK_okay";
      A     "OilLevelLow_BK";
      A     "Power_Head";
      =     "HydrBK_okay";
NETWORK
TITLE = Drucksensor Lecköl im Nachläuferaggregat
      A     "Tur";
      =     L 2.0;
      BLD   103;
      A     "Bipolar";
      =     L 2.1;
      BLD   103;
      CALL  "Scale_mts" (
           PV                       := "Pres_CaseDrain_BKAG",
           PV_high                  := 1.000000e+01,
           PV_low                   := 0.000000e+00,
           NB                       := L 2.0,
           Bipolar                  := L 2.1,
           Ueberlauf_High           := "Overflow_High",
           Ueberlauf_Low            := "Overflow_Low",
           Scaled_Value             := "DataLogging2".PresCaseDrain_BKAG);
      NOP   0;
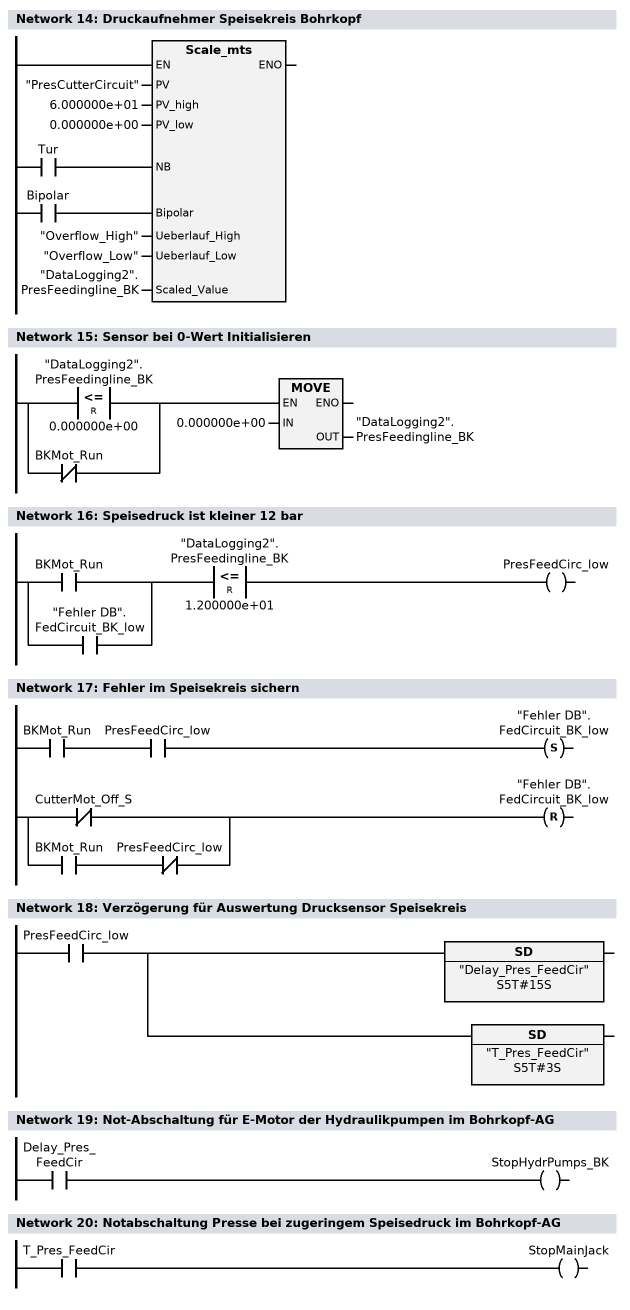
NETWORK
TITLE = Druckaufnehmer Speisekreis Bohrkopf
      A     "Tur";
      =     L 2.0;
      BLD   103;
      A     "Bipolar";
      =     L 2.1;
      BLD   103;
      CALL  "Scale_mts" (
           PV                       := "PresCutterCircuit",
           PV_high                  := 6.000000e+01,
           PV_low                   := 0.000000e+00,
           NB                       := L 2.0,
           Bipolar                  := L 2.1,
           Ueberlauf_High           := "Overflow_High",
           Ueberlauf_Low            := "Overflow_Low",
           Scaled_Value             := "DataLogging2".PresFeedingline_BK);
      NOP   0;
NETWORK
TITLE = Sensor bei 0-Wert Initialisieren
      A(;
      O(;
      L     "DataLogging2".PresFeedingline_BK;
      L     0.000000e+00;
      <=R;
      );
      ON    "BKMot_Run";
      );
      JNB   _003;
      L     0.000000e+00;
      T     "DataLogging2".PresFeedingline_BK;
_003: NOP   0;
NETWORK
TITLE = Speisedruck ist kleiner 12 bar
      A(;
      O     "BKMot_Run";
      O     "Fehler DB".FedCircuit_BK_low;
      );
      A(;
      L     "DataLogging2".PresFeedingline_BK;
      L     1.200000e+01;
      <=R;
      );
      =     "PresFeedCirc_low";
NETWORK
TITLE = Fehler im Speisekreis sichern
      A     "BKMot_Run";
      A     "PresFeedCirc_low";
      S     "Fehler DB".FedCircuit_BK_low;
      A(;
      ON    "CutterMot_Off_S";
      O;
      A     "BKMot_Run";
      AN    "PresFeedCirc_low";
      );
      R     "Fehler DB".FedCircuit_BK_low;
      NOP   0;
NETWORK
TITLE = Verzögerung für Auswertung Drucksensor Speisekreis
      A     "PresFeedCirc_low";
      L     S5T#15S;
      SD    "Delay_Pres_FeedCir";
      L     S5T#3S;
      SD    "T_Pres_FeedCir";
NETWORK
TITLE = Not-Abschaltung für E-Motor der Hydraulikpumpen im Bohrkopf-AG
      A     "Delay_Pres_FeedCir";
      =     "StopHydrPumps_BK";
NETWORK
TITLE = Notabschaltung Presse bei zugeringem Speisedruck im Bohrkopf-AG
      A     "T_Pres_FeedCir";
      =     "StopMainJack";
END_FUNCTION

FUNCTION "Filter power pack" : VOID	// FC 33
TITLE = Hydraulikölfilter im Containeraggregat
AUTHOR : Simdon
FAMILY : Freigabe
NAME : FilterPP
VERSION : 0.1
VAR_TEMP
  Ret1 : WORD ;
  Ret2 : WORD ;
  Ret3 : WORD ;
END_VAR
BEGIN
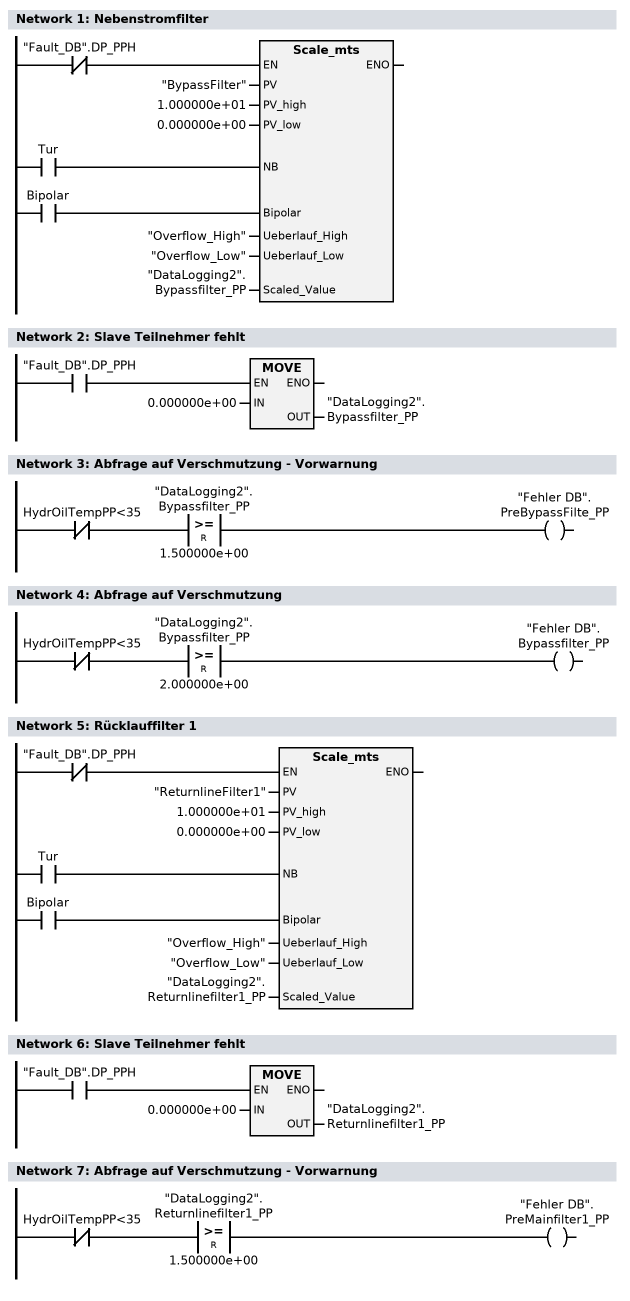
NETWORK
TITLE = Nebenstromfilter
      A     "Tur";
      =     L 6.0;
      BLD   103;
      A     "Bipolar";
      =     L 6.1;
      BLD   103;
      AN    "Fault_DB".DP_PPH;
      JNB   _001;
      CALL  "Scale_mts" (
           PV                       := "BypassFilter",
           PV_high                  := 1.000000e+01,
           PV_low                   := 0.000000e+00,
           NB                       := L 6.0,
           Bipolar                  := L 6.1,
           Ueberlauf_High           := "Overflow_High",
           Ueberlauf_Low            := "Overflow_Low",
           Scaled_Value             := "DataLogging2".Bypassfilter_PP);
_001: NOP   0;
NETWORK
TITLE = Slave Teilnehmer fehlt
      A     "Fault_DB".DP_PPH;
      JNB   _002;
      L     0.000000e+00;
      T     "DataLogging2".Bypassfilter_PP;
_002: NOP   0;
NETWORK
TITLE = Abfrage auf Verschmutzung - Vorwarnung
      AN    "HydrOilTempPP<35";
      A(;
      L     "DataLogging2".Bypassfilter_PP;
      L     1.500000e+00;
      >=R;
      );
      =     "Fehler DB".PreBypassFilte_PP;
NETWORK
TITLE = Abfrage auf Verschmutzung
      AN    "HydrOilTempPP<35";
      A(;
      L     "DataLogging2".Bypassfilter_PP;
      L     2.000000e+00;
      >=R;
      );
      =     "Fehler DB".Bypassfilter_PP;
NETWORK
TITLE = Rücklauffilter 1
      A     "Tur";
      =     L 6.0;
      BLD   103;
      A     "Bipolar";
      =     L 6.1;
      BLD   103;
      AN    "Fault_DB".DP_PPH;
      JNB   _003;
      CALL  "Scale_mts" (
           PV                       := "ReturnlineFilter1",
           PV_high                  := 1.000000e+01,
           PV_low                   := 0.000000e+00,
           NB                       := L 6.0,
           Bipolar                  := L 6.1,
           Ueberlauf_High           := "Overflow_High",
           Ueberlauf_Low            := "Overflow_Low",
           Scaled_Value             := "DataLogging2".Returnlinefilter1_PP);
_003: NOP   0;
NETWORK
TITLE = Slave Teilnehmer fehlt
      A     "Fault_DB".DP_PPH;
      JNB   _004;
      L     0.000000e+00;
      T     "DataLogging2".Returnlinefilter1_PP;
_004: NOP   0;
NETWORK
TITLE = Abfrage auf Verschmutzung - Vorwarnung
      AN    "HydrOilTempPP<35";
      A(;
      L     "DataLogging2".Returnlinefilter1_PP;
      L     1.500000e+00;
      >=R;
      );
      =     "Fehler DB".PreMainfilter1_PP;
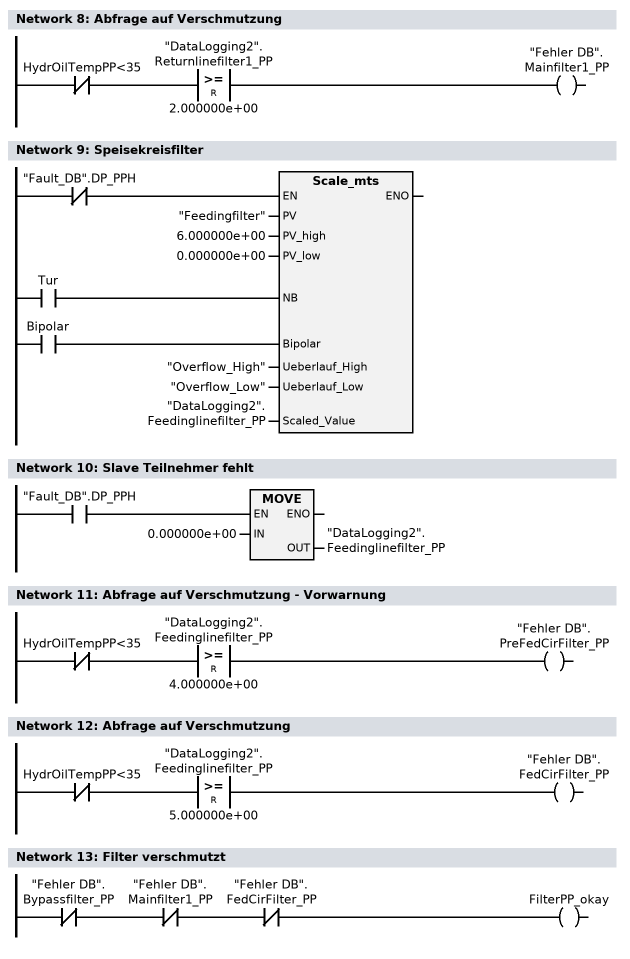
NETWORK
TITLE = Abfrage auf Verschmutzung
      AN    "HydrOilTempPP<35";
      A(;
      L     "DataLogging2".Returnlinefilter1_PP;
      L     2.000000e+00;
      >=R;
      );
      =     "Fehler DB".Mainfilter1_PP;
NETWORK
TITLE = Speisekreisfilter
      A     "Tur";
      =     L 6.0;
      BLD   103;
      A     "Bipolar";
      =     L 6.1;
      BLD   103;
      AN    "Fault_DB".DP_PPH;
      JNB   _005;
      CALL  "Scale_mts" (
           PV                       := "Feedingfilter",
           PV_high                  := 6.000000e+00,
           PV_low                   := 0.000000e+00,
           NB                       := L 6.0,
           Bipolar                  := L 6.1,
           Ueberlauf_High           := "Overflow_High",
           Ueberlauf_Low            := "Overflow_Low",
           Scaled_Value             := "DataLogging2".Feedinglinefilter_PP);
_005: NOP   0;
NETWORK
TITLE = Slave Teilnehmer fehlt
      A     "Fault_DB".DP_PPH;
      JNB   _006;
      L     0.000000e+00;
      T     "DataLogging2".Feedinglinefilter_PP;
_006: NOP   0;
NETWORK
TITLE = Abfrage auf Verschmutzung - Vorwarnung
      AN    "HydrOilTempPP<35";
      A(;
      L     "DataLogging2".Feedinglinefilter_PP;
      L     4.000000e+00;
      >=R;
      );
      =     "Fehler DB".PreFedCirFilter_PP;
NETWORK
TITLE = Abfrage auf Verschmutzung
      AN    "HydrOilTempPP<35";
      A(;
      L     "DataLogging2".Feedinglinefilter_PP;
      L     5.000000e+00;
      >=R;
      );
      =     "Fehler DB".FedCirFilter_PP;
NETWORK
TITLE = Filter verschmutzt
      AN    "Fehler DB".Bypassfilter_PP;
      AN    "Fehler DB".Mainfilter1_PP;
      AN    "Fehler DB".FedCirFilter_PP;
      =     "FilterPP_okay";
END_FUNCTION

FUNCTION "Filter_BK" : VOID	// FC 34
TITLE = Hydrauliölfilter im Bohrkopfaggregat
AUTHOR : Simdon
FAMILY : Freigabe
NAME : FilterBK
VERSION : 0.1
VAR_TEMP
  SensFedCircCutter1 : BOOL ;
  ReturnlinefilterBK : BOOL ;
END_VAR
BEGIN
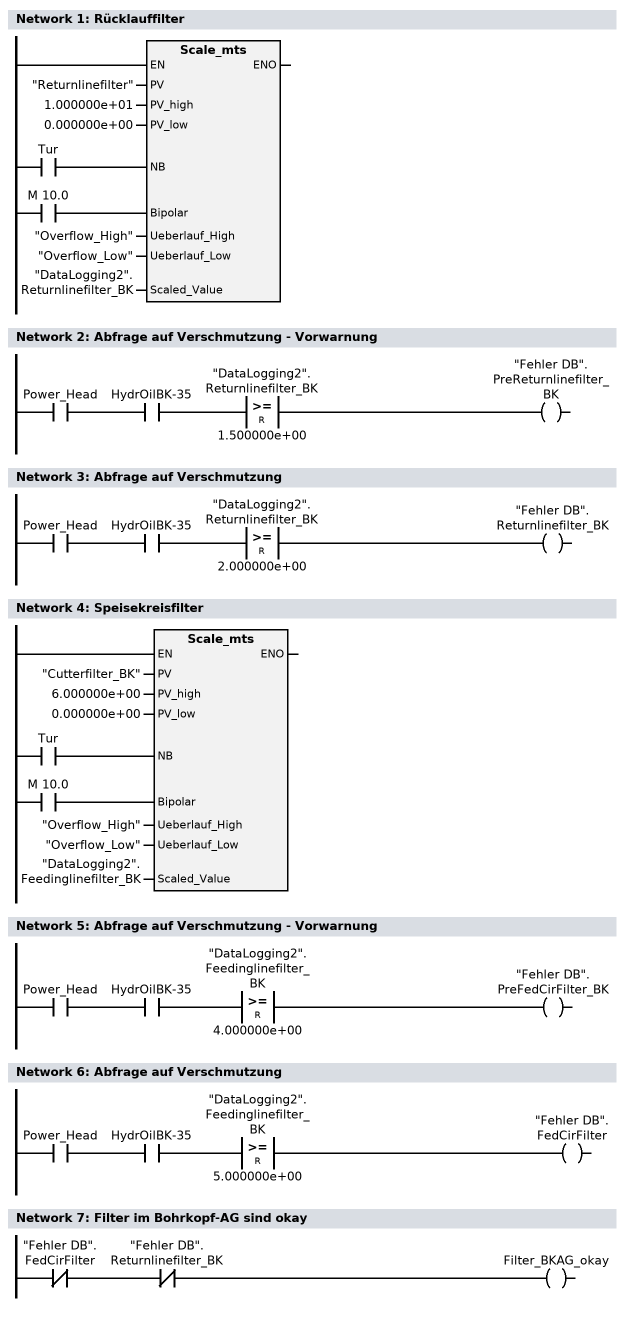
NETWORK
TITLE = Rücklauffilter
      A     "Tur";
      =     L 1.0;
      BLD   103;
      A     M 10.0;
      =     L 1.1;
      BLD   103;
      CALL  "Scale_mts" (
           PV                       := "Returnlinefilter",
           PV_high                  := 1.000000e+01,
           PV_low                   := 0.000000e+00,
           NB                       := L 1.0,
           Bipolar                  := L 1.1,
           Ueberlauf_High           := "Overflow_High",
           Ueberlauf_Low            := "Overflow_Low",
           Scaled_Value             := "DataLogging2".Returnlinefilter_BK);
      NOP   0;
NETWORK
TITLE = Abfrage auf Verschmutzung - Vorwarnung
      A     "Power_Head";
      A     "HydrOilBK-35";
      A(;
      L     "DataLogging2".Returnlinefilter_BK;
      L     1.500000e+00;
      >=R;
      );
      =     "Fehler DB".PreReturnlinefilter_BK;
NETWORK
TITLE = Abfrage auf Verschmutzung
      A     "Power_Head";
      A     "HydrOilBK-35";
      A(;
      L     "DataLogging2".Returnlinefilter_BK;
      L     2.000000e+00;
      >=R;
      );
      =     "Fehler DB".Returnlinefilter_BK;
NETWORK
TITLE = Speisekreisfilter
      A     "Tur";
      =     L 1.0;
      BLD   103;
      A     M 10.0;
      =     L 1.1;
      BLD   103;
      CALL  "Scale_mts" (
           PV                       := "Cutterfilter_BK",
           PV_high                  := 6.000000e+00,
           PV_low                   := 0.000000e+00,
           NB                       := L 1.0,
           Bipolar                  := L 1.1,
           Ueberlauf_High           := "Overflow_High",
           Ueberlauf_Low            := "Overflow_Low",
           Scaled_Value             := "DataLogging2".Feedinglinefilter_BK);
      NOP   0;
NETWORK
TITLE = Abfrage auf Verschmutzung - Vorwarnung
      A     "Power_Head";
      A     "HydrOilBK-35";
      A(;
      L     "DataLogging2".Feedinglinefilter_BK;
      L     4.000000e+00;
      >=R;
      );
      =     "Fehler DB".PreFedCirFilter_BK;
NETWORK
TITLE = Abfrage auf Verschmutzung
      A     "Power_Head";
      A     "HydrOilBK-35";
      A(;
      L     "DataLogging2".Feedinglinefilter_BK;
      L     5.000000e+00;
      >=R;
      );
      =     "Fehler DB".FedCirFilter;
NETWORK
TITLE = Filter im Bohrkopf-AG sind okay
      AN    "Fehler DB".FedCirFilter;
      AN    "Fehler DB".Returnlinefilter_BK;
      =     "Filter_BKAG_okay";
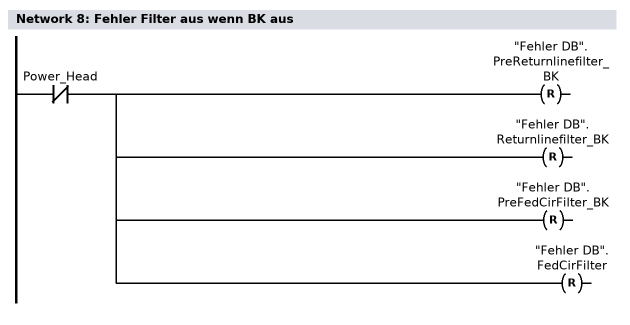
NETWORK
TITLE = Fehler Filter aus wenn BK aus
      AN    "Power_Head";
      R     "Fehler DB".PreReturnlinefilter_BK;
      R     "Fehler DB".Returnlinefilter_BK;
      R     "Fehler DB".PreFedCirFilter_BK;
      R     "Fehler DB".FedCirFilter;
END_FUNCTION

FUNCTION "Distance wheel" : VOID	// FC 35
TITLE = Messung der Vortriebslänge und Geschwindigkeit
AUTHOR : Simdon
FAMILY : Control
NAME : Distance
VERSION : 0.1
VAR_TEMP
  I_Kom : BYTE ;
  iREG_RD_ADR : INT ;
  KOM_D1 : BOOL ;
  KOM_STS_DBP1 : BOOL ;
  KOM_D2 : BOOL ;
  KOM_STS_DBP2 : BOOL ;
  KOM_STS_CONFIG_ERR : BOOL ;
  KOM_REG_RD_ABORT : BOOL ;
  KOM_REG_WR_AKN : BOOL ;
  KOM_REG_WR_ACCEPT : BOOL ;
  Schreiben : BOOL ;
  Speed_1 : REAL ;
  Speed_2 : REAL ;
  Calc1 : BOOL ;
  Calc2 : BOOL ;
END_VAR
BEGIN
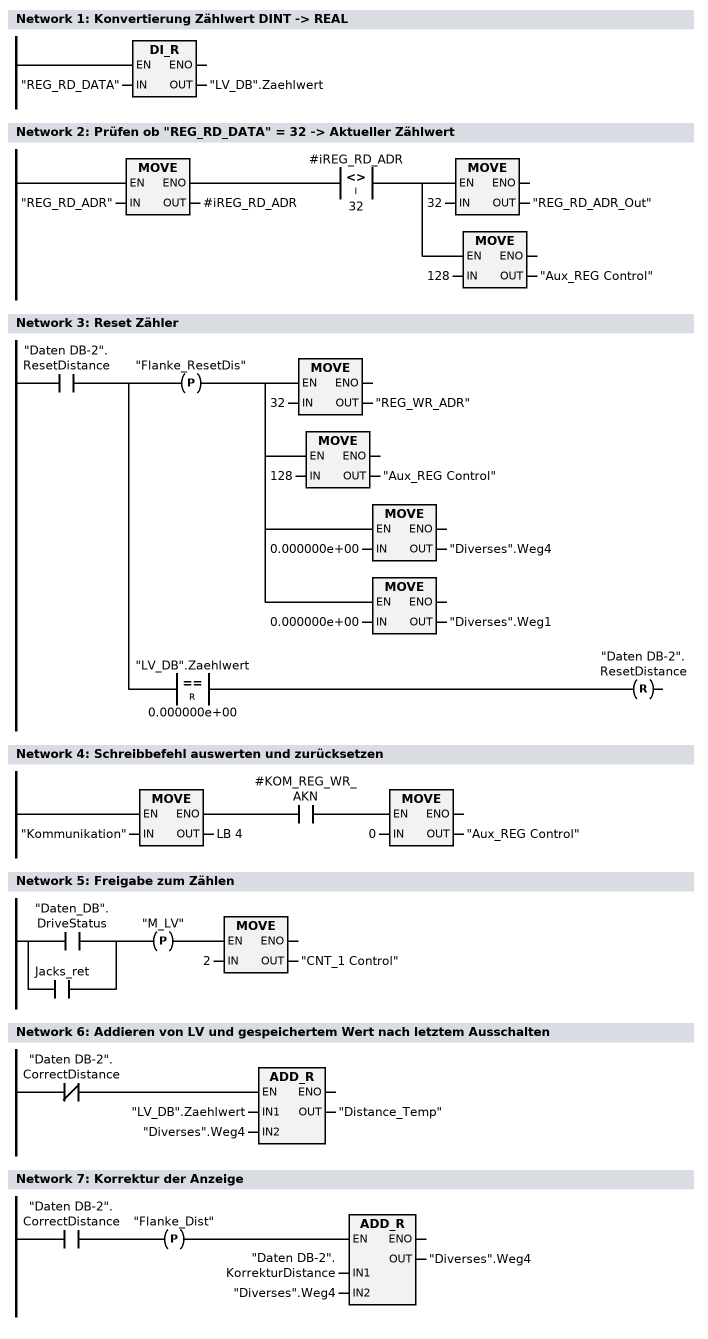
NETWORK
TITLE = Konvertierung Zählwert DINT -> REAL
      L     "REG_RD_DATA";
      DTR;
      T     "LV_DB".Zaehlwert;
      NOP   0;
NETWORK
TITLE = Prüfen ob "REG_RD_DATA" = 32 -> Aktueller Zählwert
      A(;
      L     "REG_RD_ADR";
      T     #iREG_RD_ADR;
      SET;
      SAVE;
      CLR;
      A     BR;
      );
      A(;
      L     #iREG_RD_ADR;
      L     32;
      <>I;
      );
      =     L 15.0;
      A     L 15.0;
      JNB   _001;
      L     32;
      T     "REG_RD_ADR_Out";
_001: NOP   0;
      A     L 15.0;
      JNB   _002;
      L     128;
      T     "Aux_REG Control";
_002: NOP   0;
NETWORK
TITLE = Reset Zähler
      A     "Daten DB-2".ResetDistance;
      =     L 15.0;
      A     L 15.0;
      FP    "Flanke_ResetDis";
      =     L 15.1;
      A     L 15.1;
      JNB   _003;
      L     32;
      T     "REG_WR_ADR";
_003: NOP   0;
      A     L 15.1;
      JNB   _004;
      L     128;
      T     "Aux_REG Control";
_004: NOP   0;
      A     L 15.1;
      JNB   _005;
      L     0.000000e+00;
      T     "Diverses".Weg4;
_005: NOP   0;
      A     L 15.1;
      JNB   _006;
      L     0.000000e+00;
      T     "Diverses".Weg1;
_006: NOP   0;
      A     L 15.0;
      A(;
      L     "LV_DB".Zaehlwert;
      L     0.000000e+00;
      ==R;
      );
      R     "Daten DB-2".ResetDistance;
NETWORK
TITLE = Schreibbefehl auswerten und zurücksetzen
      A(;
      L     "Kommunikation";
      T     LB 4;
      SET;
      SAVE;
      CLR;
      A     BR;
      );
      A     #KOM_REG_WR_AKN;
      JNB   _007;
      L     0;
      T     "Aux_REG Control";
_007: NOP   0;
NETWORK
TITLE = Freigabe zum Zählen
      A(;
      O     "Daten_DB".DriveStatus;
      O     "Jacks_ret";
      );
      FP    "M_LV";
      JNB   _008;
      L     2;
      T     "CNT_1 Control";
_008: NOP   0;
NETWORK
TITLE = Addieren von LV und gespeichertem Wert nach letztem Ausschalten
      AN    "Daten DB-2".CorrectDistance;
      JNB   _009;
      L     "LV_DB".Zaehlwert;
      L     "Diverses".Weg4;
      +R;
      T     "Distance_Temp";
_009: NOP   0;
NETWORK
TITLE = Korrektur der Anzeige
      A     "Daten DB-2".CorrectDistance;
      FP    "Flanke_Dist";
      JNB   _00a;
      L     "Daten DB-2".KorrekturDistance;
      L     "Diverses".Weg4;
      +R;
      T     "Diverses".Weg4;
_00a: NOP   0;
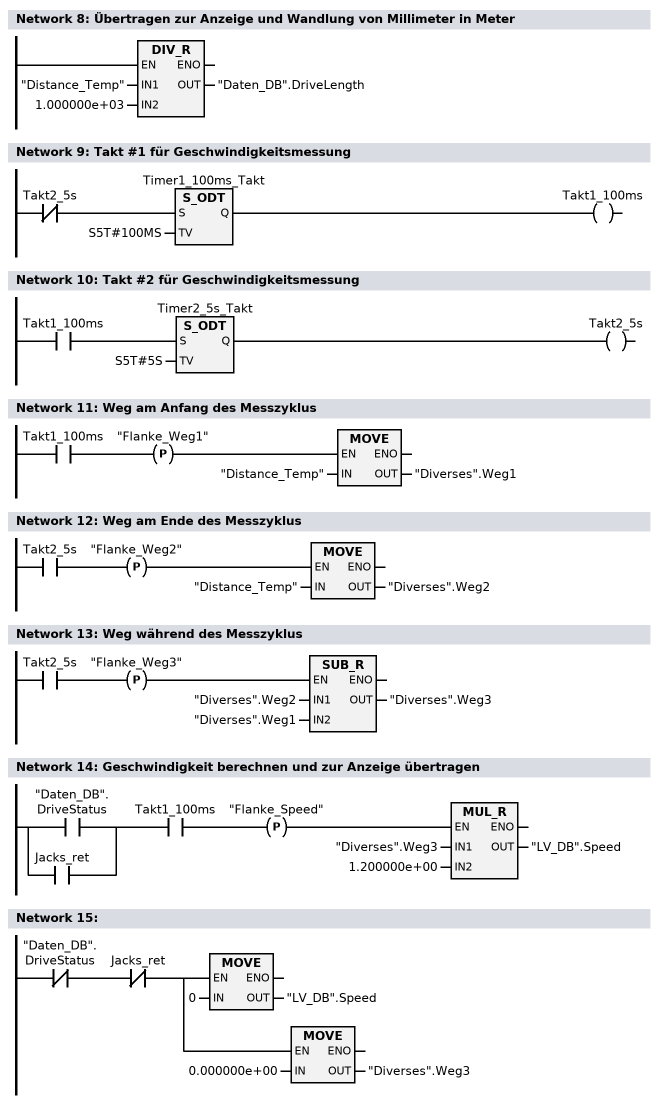
NETWORK
TITLE = Übertragen zur Anzeige und Wandlung von Millimeter in Meter
      L     "Distance_Temp";
      L     1.000000e+03;
      /R;
      T     "Daten_DB".DriveLength;
      NOP   0;
NETWORK
TITLE = Takt #1 für Geschwindigkeitsmessung
      AN    "Takt2_5s";
      L     S5T#100MS;
      SD    "Timer1_100ms_Takt";
      NOP   0;
      NOP   0;
      NOP   0;
      A     "Timer1_100ms_Takt";
      =     "Takt1_100ms";
NETWORK
TITLE = Takt #2 für Geschwindigkeitsmessung
      A     "Takt1_100ms";
      L     S5T#5S;
      SD    "Timer2_5s_Takt";
      NOP   0;
      NOP   0;
      NOP   0;
      A     "Timer2_5s_Takt";
      =     "Takt2_5s";
NETWORK
TITLE = Weg am Anfang des Messzyklus
      A     "Takt1_100ms";
      FP    "Flanke_Weg1";
      JNB   _00b;
      L     "Distance_Temp";
      T     "Diverses".Weg1;
_00b: NOP   0;
NETWORK
TITLE = Weg am Ende des Messzyklus
      A     "Takt2_5s";
      FP    "Flanke_Weg2";
      JNB   _00c;
      L     "Distance_Temp";
      T     "Diverses".Weg2;
_00c: NOP   0;
NETWORK
TITLE = Weg während des Messzyklus
      A     "Takt2_5s";
      FP    "Flanke_Weg3";
      JNB   _00d;
      L     "Diverses".Weg2;
      L     "Diverses".Weg1;
      -R;
      T     "Diverses".Weg3;
_00d: NOP   0;
NETWORK
TITLE = Geschwindigkeit berechnen und zur Anzeige übertragen
      A(;
      O     "Daten_DB".DriveStatus;
      O     "Jacks_ret";
      );
      A     "Takt1_100ms";
      FP    "Flanke_Speed";
      JNB   _00e;
      L     "Diverses".Weg3;
      L     1.200000e+00;
      *R;
      T     "LV_DB".Speed;
_00e: NOP   0;
NETWORK
TITLE =
      AN    "Daten_DB".DriveStatus;
      AN    "Jacks_ret";
      =     L 15.0;
      A     L 15.0;
      JNB   _00f;
      L     0;
      T     "LV_DB".Speed;
_00f: NOP   0;
      A     L 15.0;
      JNB   _010;
      L     0.000000e+00;
      T     "Diverses".Weg3;
_010: NOP   0;
END_FUNCTION

FUNCTION "Head" : VOID	// FC 36
TITLE = Diverses Kopf und Nachläufer
AUTHOR : Simdon
FAMILY : Head
NAME : Head
VERSION : 0.1
VAR_TEMP
  CaseDrain : BOOL ;
  HeadRoll_left : BOOL ;
  HeadRoll_right : BOOL ;
  RetVal_1 : BOOL ;
END_VAR
BEGIN
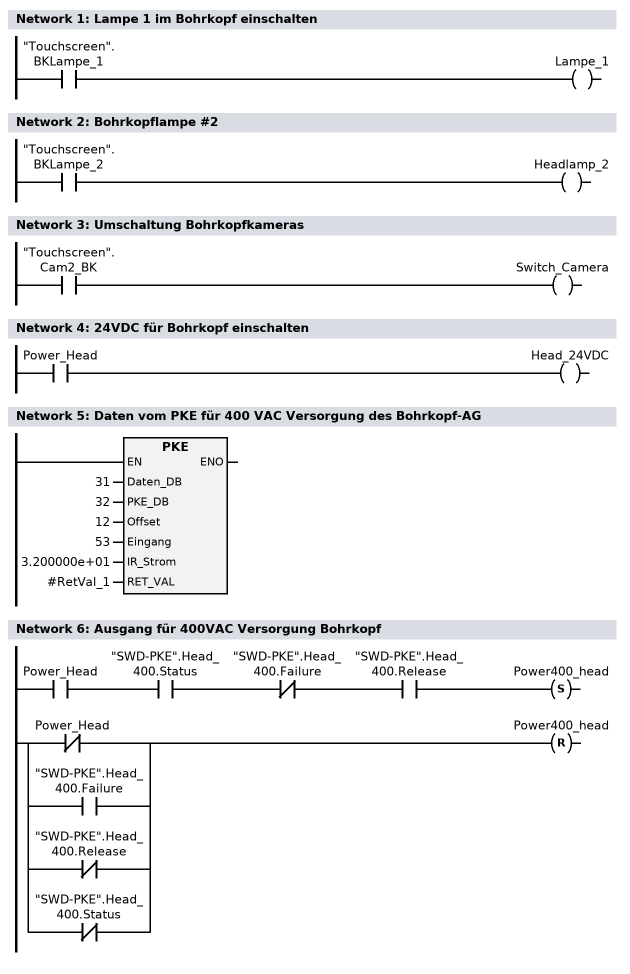
NETWORK
TITLE = Lampe 1 im Bohrkopf einschalten
      A     "Touchscreen".BKLampe_1;
      =     "Lampe_1";
NETWORK
TITLE = Bohrkopflampe #2
      A     "Touchscreen".BKLampe_2;
      =     "Headlamp_2";
NETWORK
TITLE = Umschaltung Bohrkopfkameras
      A     "Touchscreen".Cam2_BK;
      =     "Switch_Camera";
NETWORK
TITLE = 24VDC für Bohrkopf einschalten
      A     "Power_Head";
      =     "Head_24VDC";
NETWORK
TITLE = Daten vom PKE für 400 VAC Versorgung des Bohrkopf-AG
      CALL  "PKE" (
           Daten_DB                 := 31,
           PKE_DB                   := 32,
           Offset                   := 12,
           Eingang                  := 53,
           IR_Strom                 := 3.200000e+01,
           RET_VAL                  := #RetVal_1);
      NOP   0;
NETWORK
TITLE = Ausgang für 400VAC Versorgung Bohrkopf
      A     "Power_Head";
      A     "SWD-PKE".Head_400.Status;
      AN    "SWD-PKE".Head_400.Failure;
      A     "SWD-PKE".Head_400.Release;
      S     "Power400_head";
      A(;
      ON    "Power_Head";
      O     "SWD-PKE".Head_400.Failure;
      ON    "SWD-PKE".Head_400.Release;
      ON    "SWD-PKE".Head_400.Status;
      );
      R     "Power400_head";
      NOP   0;
END_FUNCTION

FUNCTION "CaseDrain" : VOID	// FC 37
TITLE = Auswertung von Lecköldruck -und sensor
AUTHOR : Simdon
FAMILY : Head
NAME : Leckoel
VERSION : 0.1
VAR_TEMP
  CaseDrain : BOOL ;
  HeadRoll_left : BOOL ;
  HeadRoll_right : BOOL ;
END_VAR
BEGIN
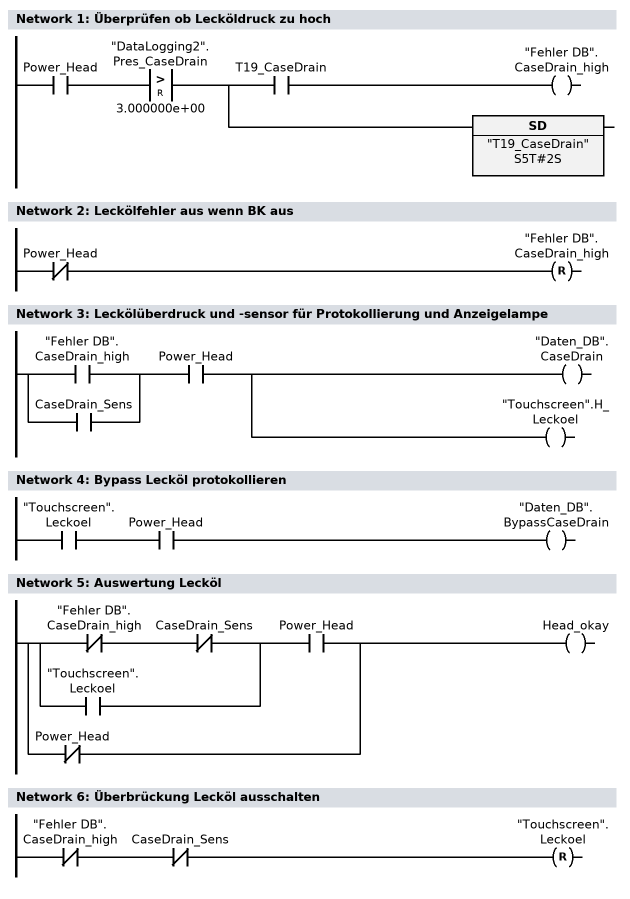
NETWORK
TITLE = Überprüfen ob Lecköldruck zu hoch
      A     "Power_Head";
      A(;
      L     "DataLogging2".Pres_CaseDrain;
      L     3.000000e+00;
      >R;
      );
      =     L 1.0;
      A     L 1.0;
      A     "T19_CaseDrain";
      =     "Fehler DB".CaseDrain_high;
      A     L 1.0;
      BLD   102;
      L     S5T#2S;
      SD    "T19_CaseDrain";
NETWORK
TITLE = Leckölfehler aus wenn BK aus
      AN    "Power_Head";
      R     "Fehler DB".CaseDrain_high;
NETWORK
TITLE = Leckölüberdruck und -sensor für Protokollierung und Anzeigelampe
      A(;
      O     "Fehler DB".CaseDrain_high;
      O     "CaseDrain_Sens";
      );
      A     "Power_Head";
      =     "Daten_DB".CaseDrain;
      =     "Touchscreen".H_Leckoel;
NETWORK
TITLE = Bypass Lecköl protokollieren
      A     "Touchscreen".Leckoel;
      A     "Power_Head";
      =     "Daten_DB".BypassCaseDrain;
NETWORK
TITLE = Auswertung Lecköl
      A(;
      AN    "Fehler DB".CaseDrain_high;
      AN    "CaseDrain_Sens";
      O     "Touchscreen".Leckoel;
      );
      A     "Power_Head";
      ON    "Power_Head";
      =     "Head_okay";
NETWORK
TITLE = Überbrückung Lecköl ausschalten
      AN    "Fehler DB".CaseDrain_high;
      AN    "CaseDrain_Sens";
      R     "Touchscreen".Leckoel;
END_FUNCTION

FUNCTION "RPM cutter" : VOID	// FC 38
TITLE = Drehzahlerfassung der Schürfscheibe
AUTHOR : Simdon
FAMILY : Head
NAME : RPM
VERSION : 0.1
VAR_TEMP
  Temp1 : REAL ;
  ReturnRead : INT ;
  ReturnWrite : INT ;
  RPM_Null : BOOL ;
END_VAR
BEGIN
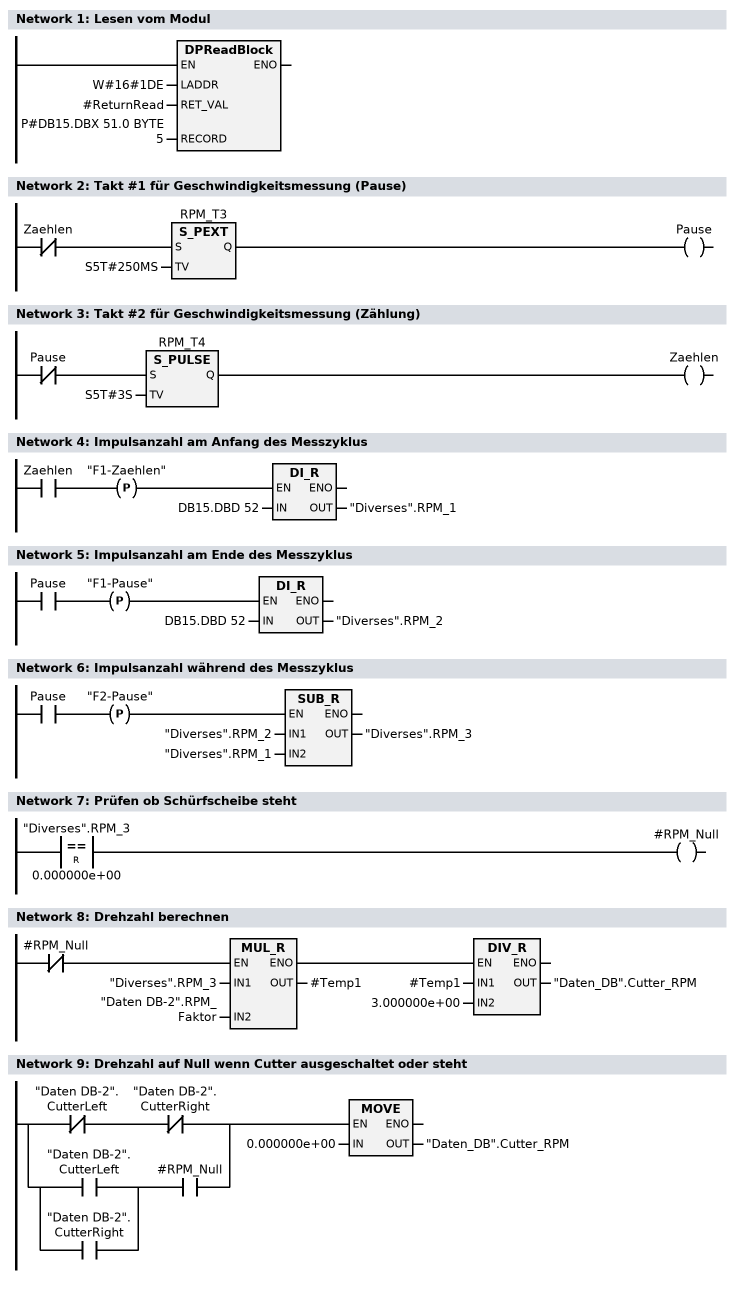
NETWORK
TITLE = Lesen vom Modul
      CALL  "DPReadBlock" (
           LADDR                    := W#16#1DE,
           RET_VAL                  := #ReturnRead,
           RECORD                   := P#DB15.DBX 51.0 BYTE 5);
      NOP   0;
NETWORK
TITLE = Takt #1 für Geschwindigkeitsmessung (Pause)
      AN    "Zaehlen";
      L     S5T#250MS;
      SE    "RPM_T3";
      NOP   0;
      NOP   0;
      NOP   0;
      A     "RPM_T3";
      =     "Pause";
NETWORK
TITLE = Takt #2 für Geschwindigkeitsmessung (Zählung)
      AN    "Pause";
      L     S5T#3S;
      SP    "RPM_T4";
      NOP   0;
      NOP   0;
      NOP   0;
      A     "RPM_T4";
      =     "Zaehlen";
NETWORK
TITLE = Impulsanzahl am Anfang des Messzyklus
      A     "Zaehlen";
      FP    "F1-Zaehlen";
      JNB   _001;
      L     DB15.DBD 52;
      DTR;
      T     "Diverses".RPM_1;
_001: NOP   0;
NETWORK
TITLE = Impulsanzahl am Ende des Messzyklus
      A     "Pause";
      FP    "F1-Pause";
      JNB   _002;
      L     DB15.DBD 52;
      DTR;
      T     "Diverses".RPM_2;
_002: NOP   0;
NETWORK
TITLE = Impulsanzahl während des Messzyklus
      A     "Pause";
      FP    "F2-Pause";
      JNB   _003;
      L     "Diverses".RPM_2;
      L     "Diverses".RPM_1;
      -R;
      T     "Diverses".RPM_3;
_003: NOP   0;
NETWORK
TITLE = Prüfen ob Schürfscheibe steht
      L     "Diverses".RPM_3;
      L     0.000000e+00;
      ==R;
      =     #RPM_Null;
NETWORK
TITLE = Drehzahl berechnen
//Der Multiplikator entspricht der max. Impulszahl pro Umdrehung korrigiert um 
//den 
//Zeitfaktor für die Umrechung Sekunden auf Minuten (60/max. Impulszahl)
//Der Divisor entspricht der Zeit für die Impulszählung.
      A(;
      AN    #RPM_Null;
      JNB   _004;
      L     "Diverses".RPM_3;
      L     "Daten DB-2".RPM_Faktor;
      *R;
      T     #Temp1;
      AN    OV;
      SAVE;
      CLR;
_004: A     BR;
      );
      JNB   _005;
      L     #Temp1;
      L     3.000000e+00;
      /R;
      T     "Daten_DB".Cutter_RPM;
_005: NOP   0;
NETWORK
TITLE = Drehzahl auf Null wenn Cutter ausgeschaltet oder steht
      A(;
      AN    "Daten DB-2".CutterLeft;
      AN    "Daten DB-2".CutterRight;
      O;
      A(;
      O     "Daten DB-2".CutterLeft;
      O     "Daten DB-2".CutterRight;
      );
      A     #RPM_Null;
      );
      JNB   _006;
      L     0.000000e+00;
      T     "Daten_DB".Cutter_RPM;
_006: NOP   0;
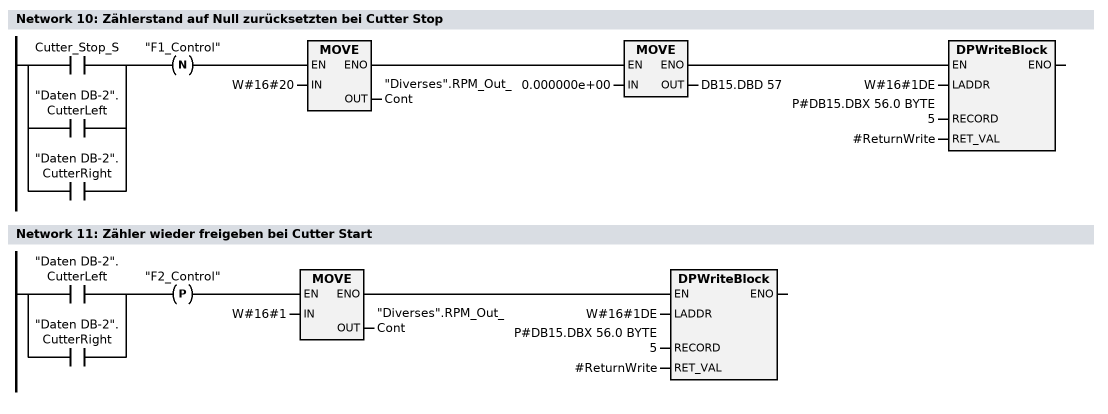
NETWORK
TITLE = Zählerstand auf Null zurücksetzten bei Cutter Stop
      A(;
      A(;
      A(;
      O     "Cutter_Stop_S";
      O     "Daten DB-2".CutterLeft;
      O     "Daten DB-2".CutterRight;
      );
      FN    "F1_Control";
      JNB   _007;
      L     W#16#20;
      T     "Diverses".RPM_Out_Cont;
      SET;
      SAVE;
      CLR;
_007: A     BR;
      );
      JNB   _008;
      L     0.000000e+00;
      T     DB15.DBD 57;
      SET;
      SAVE;
      CLR;
_008: A     BR;
      );
      JNB   _009;
      CALL  "DPWriteBlock" (
           LADDR                    := W#16#1DE,
           RECORD                   := P#DB15.DBX 56.0 BYTE 5,
           RET_VAL                  := #ReturnWrite);
_009: NOP   0;
NETWORK
TITLE = Zähler wieder freigeben bei Cutter Start
      A(;
      A(;
      O     "Daten DB-2".CutterLeft;
      O     "Daten DB-2".CutterRight;
      );
      FP    "F2_Control";
      JNB   _00a;
      L     W#16#1;
      T     "Diverses".RPM_Out_Cont;
      SET;
      SAVE;
      CLR;
_00a: A     BR;
      );
      JNB   _00b;
      CALL  "DPWriteBlock" (
           LADDR                    := W#16#1DE,
           RECORD                   := P#DB15.DBX 56.0 BYTE 5,
           RET_VAL                  := #ReturnWrite);
_00b: NOP   0;
END_FUNCTION

FUNCTION "PresSensor_BK" : VOID	// FC 39
TITLE = Drucksensoren über Piconet im Bohrkopf
AUTHOR : Simdon
FAMILY : BK
NAME : PresBK
VERSION : 0.1
BEGIN
